KUKA KRL program: MyProgram_253().src

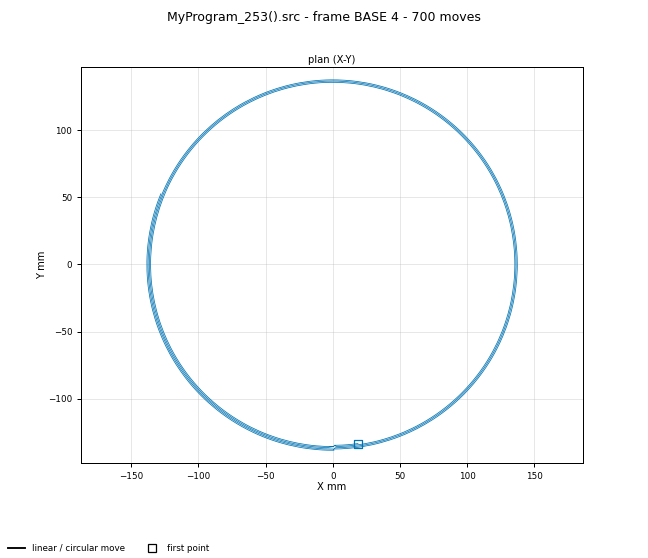
[picture p0: tool path of MyProgram_253().src in frame BASE 4, 700 of 700 moves have a stored position in this frame; points joined in program order, loops and branches not executed]
&ACCESS RVP
&REL 1
&PARAM TEMPLATE = C:\KRC\Roboter\Template\vorgabe
&PARAM EDITMASK = *
DEF MyProgram_253()
; ---- Setting reference (Base) ----
$BASE = BASE_DATA[4]

; --------------------------
; ---- Setting tool (TCP) ----
$TOOL = TOOL_DATA[3]
; --------------------------

$VEL.CP = VEL_APROX_PRINT
Startdeposition()
$VEL.CP = VEL_PRINT
LIN {X 18.8097,Y -133.4108,Z 165,A -80.9868,B 11.6438,C 0.2776,E1 11.6692,E2 531.5749} C_DIS
LIN {X 14.6629,Y -133.9301,Z 165,A -82.8153,B 11.6437,C 0.2797,E1 11.6641,E2 533.4109} C_DIS
LIN {X 11.2061,Y -134.2633,Z 165,A -84.2006,B 11.6437,C 0.278,E1 11.6603,E2 534.7857} C_DIS
LIN {X 7.424,Y -134.5271,Z 165,A -85.9426,B 11.6437,C 0.2818,E1 11.6554,E2 536.5447} C_DIS
LIN {X 3.6896,Y -134.6797,Z 165,A -87.3882,B 11.6437,C 0.2785,E1 11.6514,E2 537.9732} C_DIS
LIN {X 0.9754,Y -134.7225,Z 165,A -88.2258,B 11.6439,C 0.2708,E1 11.6492,E2 538.7721} C_DIS
Enddeposition()
LIN {X 0.9754,Y -134.7225,Z 165,A -88.2258,B 11.6439,C 0.2708,E1 11.6492,E2 538.7721} C_DIS
Startdeposition()
$VEL.CP = VEL_PRINT
LIN {X 3.0109,Y -135.617,Z 165,A -86.906,B 11.5615,C 0.2702,E1 11.5704,E2 537.4539} C_DIS
LIN {X 6.5276,Y -135.4914,Z 165,A -85.4969,B 11.5615,C 0.2718,E1 11.5743,E2 536.0536} C_DIS
LIN {X 10.0387,Y -135.2764,Z 165,A -84.0037,B 11.5615,C 0.2711,E1 11.5785,E2 534.5587} C_DIS
LIN {X 14.2252,Y -134.9006,Z 165,A -82.4774,B 11.5613,C 0.2767,E1 11.5827,E2 533.0628} C_DIS
LIN {X 17.3372,Y -134.536,Z 165,A -80.9699,B 11.5615,C 0.2714,E1 11.5869,E2 531.5314} C_DIS
LIN {X 20.6164,Y -134.0724,Z 165,A -79.5566,B 11.5615,C 0.2702,E1 11.5908,E2 530.1154} C_DIS
LIN {X 24.6834,Y -133.3858,Z 165,A -77.688,B 11.5615,C 0.2658,E1 11.596,E2 528.2297} C_DIS
LIN {X 27.8368,Y -132.7635,Z 165,A -76.3315,B 11.5616,C 0.2649,E1 11.5997,E2 526.8724} C_DIS
LIN {X 30.9968,Y -132.0615,Z 165,A -74.966,B 11.5616,C 0.2638,E1 11.6034,E2 525.5062} C_DIS
LIN {X 34.1606,Y -131.2787,Z 165,A -73.7387,B 11.5616,C 0.2666,E1 11.6067,E2 524.2967} C_DIS
LIN {X 37.6859,Y -130.3086,Z 165,A -72.3391,B 11.5616,C 0.2689,E1 11.6104,E2 522.9142} C_DIS
LIN {X 40.9847,Y -129.3086,Z 165,A -70.9423,B 11.5616,C 0.269,E1 11.6141,E2 521.5237} C_DIS
LIN {X 43.6454,Y -128.4373,Z 165,A -69.4187,B 11.5617,C 0.2588,E1 11.6183,E2 519.9563} C_DIS
LIN {X 47.2884,Y -127.1387,Z 165,A -67.9407,B 11.5617,C 0.261,E1 11.6221,E2 518.4965} C_DIS
LIN {X 49.9322,Y -126.1262,Z 165,A -66.7499,B 11.5617,C 0.2598,E1 11.6252,E2 517.3055} C_DIS
LIN {X 53.0552,Y -124.8446,Z 165,A -65.3304,B 11.5617,C 0.2581,E1 11.6289,E2 515.8856} C_DIS
LIN {X 56.4766,Y -123.3327,Z 165,A -63.8884,B 11.5617,C 0.2597,E1 11.6325,E2 514.4594} C_DIS
LIN {X 59.2442,Y -122.0294,Z 165,A -62.4727,B 11.5618,C 0.2546,E1 11.6361,E2 513.0272} C_DIS
LIN {X 62.3035,Y -120.4961,Z 165,A -60.97,B 11.5619,C 0.251,E1 11.6399,E2 511.5159} C_DIS
LIN {X 66.0881,Y -118.4627,Z 165,A -59.1023,B 11.562,C 0.2468,E1 11.6445,E2 509.6398} C_DIS
LIN {X 69.8227,Y -116.3006,Z 165,A -57.2966,B 11.562,C 0.2443,E1 11.6488,E2 507.8345} C_DIS
LIN {X 73.5009,Y -114.0116,Z 165,A -55.5367,B 11.562,C 0.2431,E1 11.6529,E2 506.0816} C_DIS
LIN {X 77.1164,Y -111.598,Z 165,A -53.6553,B 11.5622,C 0.2386,E1 11.6573,E2 504.1927} C_DIS
LIN {X 80.6628,Y -109.0622,Z 165,A -51.8858,B 11.5622,C 0.2372,E1 11.6613,E2 502.4305} C_DIS
LIN {X 84.1341,Y -106.4072,Z 165,A -50.0545,B 11.5622,C 0.2341,E1 11.6653,E2 500.5991} C_DIS
LIN {X 87.5243,Y -103.6366,Z 165,A -48.1855,B 11.5624,C 0.2299,E1 11.6693,E2 498.7257} C_DIS
LIN {X 90.8278,Y -100.7539,Z 165,A -46.385,B 11.5624,C 0.2275,E1 11.6731,E2 496.9297} C_DIS
LIN {X 93.8395,Y -97.9542,Z 165,A -44.6945,B 11.5624,C 0.2251,E1 11.6765,E2 495.2431} C_DIS
LIN {X 96.5381,Y -95.2966,Z 165,A -43.0391,B 11.5625,C 0.2201,E1 11.6798,E2 493.579} C_DIS
LIN {X 99.5704,Y -92.1237,Z 165,A -41.3104,B 11.5625,C 0.2194,E1 11.6831,E2 491.8641} C_DIS
LIN {X 101.9202,Y -89.5172,Z 165,A -39.7769,B 11.5626,C 0.2146,E1 11.6859,E2 490.3225} C_DIS
LIN {X 104.7585,Y -86.1783,Z 165,A -37.8873,B 11.5627,C 0.2092,E1 11.6893,E2 488.4259} C_DIS
LIN {X 107.563,Y -82.6508,Z 165,A -36.0363,B 11.5627,C 0.206,E1 11.6925,E2 486.5794} C_DIS
LIN {X 110.091,Y -79.2529,Z 165,A -34.2361,B 11.5629,C 0.2013,E1 11.6955,E2 484.7757} C_DIS
LIN {X 112.5783,Y -75.6781,Z 165,A -32.4181,B 11.5629,C 0.1973,E1 11.6983,E2 482.9583} C_DIS
LIN {X 115.0446,Y -71.8725,Z 165,A -30.6305,B 11.5629,C 0.196,E1 11.701,E2 481.1846} C_DIS
LIN {X 117.1808,Y -68.3353,Z 165,A -28.8018,B 11.5631,C 0.1892,E1 11.7036,E2 479.3433} C_DIS
LIN {X 119.3066,Y -64.552,Z 165,A -27.0042,B 11.5631,C 0.1853,E1 11.706,E2 477.5481} C_DIS
LIN {X 120.7405,Y -61.8235,Z 165,A -25.8285,B 11.5631,C 0.1853,E1 11.7075,E2 476.3866} C_DIS
LIN {X 122.2606,Y -58.7602,Z 165,A -24.4024,B 11.5631,C 0.182,E1 11.7093,E2 474.9612} C_DIS
LIN {X 123.609,Y -55.8697,Z 165,A -23.1901,B 11.5631,C 0.182,E1 11.7107,E2 473.7643} C_DIS
LIN {X 125.0285,Y -52.615,Z 165,A -21.5784,B 11.5633,C 0.1748,E1 11.7125,E2 472.1368} C_DIS
LIN {X 126.1262,Y -49.9322,Z 165,A -20.3839,B 11.5633,C 0.1722,E1 11.7137,E2 470.9447} C_DIS
LIN {X 127.3237,Y -46.7945,Z 165,A -18.8366,B 11.5634,C 0.1646,E1 11.7152,E2 469.3796} C_DIS
LIN {X 128.6025,Y -43.1491,Z 165,A -17.5683,B 11.5634,C 0.1702,E1 11.7163,E2 468.1549} C_DIS
LIN {X 129.6194,Y -39.9908,Z 165,A -15.9931,B 11.5634,C 0.1614,E1 11.7177,E2 466.5564} C_DIS
LIN {X 130.5534,Y -36.8277,Z 165,A -14.6194,B 11.5635,C 0.1579,E1 11.7187,E2 465.1834} C_DIS
LIN {X 131.2787,Y -34.1606,Z 165,A -13.3235,B 11.5636,C 0.151,E1 11.7197,E2 463.8702} C_DIS
LIN {X 132.0615,Y -30.9968,Z 165,A -11.9672,B 11.5636,C 0.1476,E1 11.7206,E2 462.515} C_DIS
LIN {X 132.8446,Y -27.4386,Z 165,A -10.5679,B 11.5636,C 0.147,E1 11.7214,E2 461.1313} C_DIS
LIN {X 133.4744,Y -24.1886,Z 165,A -9.216,B 11.5637,C 0.1442,E1 11.722,E2 459.7837} C_DIS
LIN {X 133.9295,Y -21.5393,Z 165,A -8.0963,B 11.5637,C 0.1414,E1 11.7226,E2 458.6648} C_DIS
LIN {X 134.4521,Y -17.9776,Z 165,A -6.5824,B 11.5638,C 0.1371,E1 11.7231,E2 457.1498} C_DIS
LIN {X 134.8403,Y -14.7856,Z 165,A -5.2517,B 11.5638,C 0.1338,E1 11.7236,E2 455.8211} C_DIS
LIN {X 135.2321,Y -10.6455,Z 165,A -3.393,B 11.5639,C 0.1258,E1 11.724,E2 453.9477} C_DIS
LIN {X 135.4388,Y -7.5745,Z 165,A -2.248,B 11.5639,C 0.1263,E1 11.7242,E2 452.8208} C_DIS
LIN {X 135.5882,Y -4.0496,Z 165,A -0.7384,B 11.5639,C 0.1214,E1 11.7244,E2 451.307} C_DIS
LIN {X 135.6518,Y -0.0881,Z 165,A 0.931,B 11.564,C 0.1166,E1 11.7244,E2 449.6365} C_DIS
LIN {X 135.617,Y 3.0109,Z 165,A 2.3297,B 11.564,C 0.1102,E1 11.7244,E2 448.2252} C_DIS
LIN {X 135.4388,Y 7.5745,Z 165,A 4.2095,B 11.5641,C 0.1059,E1 11.7241,E2 446.3495} C_DIS
LIN {X 135.1735,Y 11.3391,Z 165,A 5.6788,B 11.5641,C 0.1047,E1 11.7238,E2 444.8941} C_DIS
LIN {X 134.786,Y 15.2895,Z 165,A 7.4472,B 11.5642,C 0.0972,E1 11.7232,E2 443.1126} C_DIS
LIN {X 134.3255,Y 18.8991,Z 165,A 8.828,B 11.5642,C 0.0972,E1 11.7227,E2 441.7497} C_DIS
LIN {X 133.9295,Y 21.5393,Z 165,A 10.076,B 11.5642,C 0.0905,E1 11.7222,E2 440.4858} C_DIS
LIN {X 133.3259,Y 24.9967,Z 165,A 11.4669,B 11.5642,C 0.0888,E1 11.7215,E2 439.1048} C_DIS
LIN {X 132.7036,Y 28.1146,Z 165,A 12.7978,B 11.5642,C 0.0853,E1 11.7207,E2 437.7741} C_DIS
LIN {X 131.9194,Y 31.5863,Z 165,A 14.2211,B 11.5643,C 0.0832,E1 11.7198,E2 436.3594} C_DIS
LIN {X 130.8567,Y 35.7431,Z 165,A 16.0164,B 11.5643,C 0.0786,E1 11.7186,E2 434.5646} C_DIS
LIN {X 129.9511,Y 38.9071,Z 165,A 17.5386,B 11.5643,C 0.071,E1 11.7173,E2 433.0247} C_DIS
LIN {X 128.9627,Y 42.0675,Z 165,A 18.8807,B 11.5644,C 0.0687,E1 11.7162,E2 431.6885} C_DIS
LIN {X 127.7125,Y 45.716,Z 165,A 20.3863,B 11.5644,C 0.0676,E1 11.7148,E2 430.1967} C_DIS
LIN {X 126.5438,Y 48.8579,Z 165,A 21.5904,B 11.5644,C 0.0696,E1 11.7137,E2 429.0177} C_DIS
LIN {X 125.4959,Y 51.4958,Z 165,A 22.9728,B 11.5644,C 0.0613,E1 11.7122,E2 427.6118} C_DIS
LIN {X 124.009,Y 54.9753,Z 165,A 24.592,B 11.5644,C 0.0564,E1 11.7104,E2 425.9886} C_DIS
LIN {X 122.7647,Y 57.7051,Z 165,A 25.8078,B 11.5644,C 0.0545,E1 11.709,E2 424.7782} C_DIS
LIN {X 121.1879,Y 60.9446,Z 165,A 27.3539,B 11.5644,C 0.0499,E1 11.707,E2 423.228} C_DIS
LIN {X 119.4381,Y 64.3071,Z 165,A 28.94,B 11.5645,C 0.0462,E1 11.705,E2 421.6426} C_DIS
LIN {X 117.3168,Y 68.1004,Z 165,A 30.7505,B 11.5645,C 0.0422,E1 11.7025,E2 419.834} C_DIS
LIN {X 115.0863,Y 71.8055,Z 165,A 32.5825,B 11.5645,C 0.0376,E1 11.6998,E2 418.0002} C_DIS
LIN {X 112.9044,Y 75.1896,Z 165,A 34.3027,B 11.5645,C 0.0329,E1 11.6971,E2 416.2765} C_DIS
LIN {X 110.2505,Y 79.0298,Z 165,A 36.1948,B 11.5645,C 0.0304,E1 11.6941,E2 414.393} C_DIS
LIN {X 107.8473,Y 82.279,Z 165,A 37.9476,B 11.5645,C 0.0252,E1 11.6912,E2 412.6336} C_DIS
LIN {X 105.1384,Y 85.7135,Z 165,A 39.7777,B 11.5645,C 0.0215,E1 11.688,E2 410.8047} C_DIS
LIN {X 102.11,Y 89.2997,Z 165,A 41.6814,B 11.5645,C 0.0193,E1 11.6845,E2 408.9098} C_DIS
LIN {X 99.3823,Y 92.3257,Z 165,A 43.4086,B 11.5645,C 0.0155,E1 11.6813,E2 407.181} C_DIS
LIN {X 96.4447,Y 95.3906,Z 165,A 45.241,B 11.5645,C 0.0107,E1 11.6777,E2 405.343} C_DIS
LIN {X 93.2037,Y 98.5594,Z 165,A 47.0833,B 11.5646,C 0.0088,E1 11.674,E2 403.5088} C_DIS
LIN {X 90.0627,Y 101.4379,Z 165,A 48.9007,B 11.5646,C 0.0049,E1 11.6702,E2 401.6886} C_DIS
LIN {X 86.853,Y 104.1998,Z 165,A 50.7053,B 11.5646,C 0.0011,E1 11.6664,E2 399.8814} C_DIS
LIN {X 83.4461,Y 106.9476,Z 165,A 52.5387,B 11.5646,C -0.0017,E1 11.6623,E2 398.0494} C_DIS
LIN {X 79.9593,Y 109.579,Z 165,A 54.3106,B 11.5646,C -0.0029,E1 11.6584,E2 396.286} C_DIS
LIN {X 76.3986,Y 112.0906,Z 165,A 56.195,B 11.5646,C -0.0071,E1 11.654,E2 394.3958} C_DIS
LIN {X 72.7701,Y 114.4795,Z 165,A 57.9895,B 11.5646,C -0.0089,E1 11.6498,E2 392.6059} C_DIS
LIN {X 69.0801,Y 116.7432,Z 165,A 59.7732,B 11.5646,C -0.0104,E1 11.6456,E2 390.8275} C_DIS
LIN {X 65.335,Y 118.8797,Z 165,A 61.6147,B 11.5646,C -0.0134,E1 11.6411,E2 388.9832} C_DIS
LIN {X 61.8235,Y 120.7405,Z 165,A 63.1832,B 11.5646,C -0.0128,E1 11.6372,E2 387.428} C_DIS
LIN {X 58.7602,Y 122.2606,Z 165,A 64.6185,B 11.5646,C -0.0143,E1 11.6336,E2 385.9938} C_DIS
LIN {X 55.7713,Y 123.653,Z 165,A 65.996,B 11.5646,C -0.0156,E1 11.6302,E2 384.6182} C_DIS
LIN {X 53.0552,Y 124.8446,Z 165,A 67.2485,B 11.5646,C -0.0169,E1 11.6269,E2 383.3658} C_DIS
LIN {X 49.9322,Y 126.1262,Z 165,A 68.666,B 11.5646,C -0.0182,E1 11.6233,E2 381.9494} C_DIS
LIN {X 46.2991,Y 127.5023,Z 165,A 70.2974,B 11.5646,C -0.0196,E1 11.619,E2 380.3191} C_DIS
LIN {X 43.1491,Y 128.6025,Z 165,A 71.5042,B 11.5646,C -0.0157,E1 11.6159,E2 379.1371} C_DIS
LIN {X 39.9908,Y 129.6194,Z 165,A 73.0939,B 11.5646,C -0.0217,E1 11.6116,E2 377.5247} C_DIS
LIN {X 36.8277,Y 130.5534,Z 165,A 74.4804,B 11.5646,C -0.0225,E1 11.6079,E2 376.1392} C_DIS
LIN {X 33.5566,Y 131.432,Z 165,A 75.8775,B 11.5646,C -0.0227,E1 11.6041,E2 374.7464} C_DIS
LIN {X 30.9968,Y 132.0615,Z 165,A 77.159,B 11.5646,C -0.0276,E1 11.6006,E2 373.4448} C_DIS
LIN {X 27.2576,Y 132.8814,Z 165,A 78.6291,B 11.5646,C -0.0248,E1 11.5966,E2 371.9929} C_DIS
LIN {X 24.0786,Y 133.494,Z 165,A 79.9581,B 11.5646,C -0.0245,E1 11.593,E2 370.669} C_DIS
LIN {X 19.9716,Y 134.1722,Z 165,A 81.7388,B 11.5646,C -0.0258,E1 11.5881,E2 368.8862} C_DIS
LIN {X 16.3568,Y 134.6587,Z 165,A 83.3166,B 11.5646,C -0.0272,E1 11.5837,E2 367.3043} C_DIS
LIN {X 12.9514,Y 135.0285,Z 165,A 84.5827,B 11.5646,C -0.0231,E1 11.5802,E2 366.0606} C_DIS
LIN {X 8.6253,Y 135.3741,Z 165,A 86.3643,B 11.5646,C -0.0222,E1 11.5753,E2 364.2859} C_DIS
LIN {X 6.0473,Y 135.5156,Z 165,A 87.7701,B 11.5646,C -0.03,E1 11.5712,E2 362.8424} C_DIS
LIN {X 2.2479,Y 135.6297,Z 165,A 89.2777,B 11.5646,C -0.0276,E1 11.5671,E2 361.3474} C_DIS
LIN {X -1.5021,Y 135.6421,Z 165,A 90.821,B 11.5646,C -0.0265,E1 11.5628,E2 359.8098} C_DIS
LIN {X -5.0045,Y 135.5563,Z 165,A 92.3049,B 11.5646,C -0.0265,E1 11.5586,E2 358.3261} C_DIS
LIN {X -9.5911,Y 135.3091,Z 165,A 94.2998,B 11.5646,C -0.0273,E1 11.5531,E2 356.3256} C_DIS
LIN {X -13.0285,Y 135.0211,Z 165,A 95.7196,B 11.5646,C -0.0259,E1 11.5491,E2 354.9111} C_DIS
LIN {X -16.3568,Y 134.6587,Z 165,A 97.1764,B 11.5646,C -0.0264,E1 11.5451,E2 353.4499} C_DIS
LIN {X -20.4646,Y 134.0959,Z 165,A 98.701,B 11.5646,C -0.0201,E1 11.5409,E2 351.9539} C_DIS
LIN {X -23.5279,Y 133.5926,Z 165,A 100.0547,B 11.5646,C -0.0204,E1 11.5372,E2 350.5958} C_DIS
LIN {X -26.7552,Y 132.9836,Z 165,A 101.4078,B 11.5646,C -0.0188,E1 11.5335,E2 349.2478} C_DIS
LIN {X -29.9133,Y 132.309,Z 165,A 102.9616,B 11.5646,C -0.0223,E1 11.5292,E2 347.672} C_DIS
LIN {X -33.154,Y 131.5342,Z 165,A 104.3866,B 11.5646,C -0.0217,E1 11.5253,E2 346.2458} C_DIS
LIN {X -37.3253,Y 130.4142,Z 165,A 106.2181,B 11.5646,C -0.0203,E1 11.5204,E2 344.4148} C_DIS
LIN {X -40.9847,Y 129.3086,Z 165,A 107.6438,B 11.5646,C -0.0144,E1 11.5167,E2 343.0131} C_DIS
LIN {X -43.6454,Y 128.4373,Z 165,A 109.1827,B 11.5646,C -0.0216,E1 11.5125,E2 341.4321} C_DIS
LIN {X -47.2884,Y 127.1387,Z 165,A 110.694,B 11.5646,C -0.017,E1 11.5086,E2 339.9369} C_DIS
LIN {X -50.0761,Y 126.0682,Z 165,A 112.0495,B 11.5646,C -0.0177,E1 11.505,E2 338.571} C_DIS
LIN {X -53.5443,Y 124.6332,Z 165,A 113.5395,B 11.5646,C -0.0136,E1 11.5012,E2 337.0939} C_DIS
LIN {X -56.1603,Y 123.479,Z 165,A 114.8903,B 11.5646,C -0.0154,E1 11.4977,E2 335.7268} C_DIS
LIN {X -59.6227,Y 121.8427,Z 165,A 116.2236,B 11.5646,C -0.0067,E1 11.4945,E2 334.4294} C_DIS
LIN {X -62.3035,Y 120.4961,Z 165,A 117.7264,B 11.5646,C -0.0103,E1 11.4906,E2 332.8992} C_DIS
LIN {X -66.0881,Y 118.4627,Z 165,A 119.6134,B 11.5646,C -0.0093,E1 11.486,E2 331.005} C_DIS
LIN {X -69.8227,Y 116.3006,Z 165,A 121.4506,B 11.5646,C -0.0068,E1 11.4816,E2 329.1679} C_DIS
LIN {X -73.5009,Y 114.0116,Z 165,A 123.2364,B 11.5646,C -0.0029,E1 11.4774,E2 327.3892} C_DIS
LIN {X -77.1164,Y 111.598,Z 165,A 125.1472,B 11.5646,C -0.0014,E1 11.473,E2 325.471} C_DIS
LIN {X -80.782,Y 108.9734,Z 165,A 126.9705,B 11.5646,C 0.0038,E1 11.4689,E2 323.6595} C_DIS
LIN {X -84.1341,Y 106.4072,Z 165,A 128.8073,B 11.5646,C 0.0059,E1 11.4648,E2 321.818} C_DIS
LIN {X -87.5243,Y 103.6366,Z 165,A 130.7206,B 11.5646,C 0.008,E1 11.4607,E2 319.8989} C_DIS
LIN {X -90.9093,Y 100.6799,Z 165,A 132.5608,B 11.5646,C 0.0131,E1 11.4569,E2 318.0676} C_DIS
LIN {X -93.8395,Y 97.9542,Z 165,A 134.2643,B 11.5646,C 0.0163,E1 11.4534,E2 316.3643} C_DIS
LIN {X -96.5381,Y 95.2966,Z 165,A 135.9106,B 11.5646,C 0.0187,E1 11.4502,E2 314.7141} C_DIS
LIN {X -99.5589,Y 92.136,Z 165,A 137.8243,B 11.5646,C 0.0213,E1 11.4465,E2 312.7943} C_DIS
LIN {X -102.4967,Y 88.8564,Z 165,A 139.7132,B 11.5646,C 0.0248,E1 11.443,E2 310.9038} C_DIS
LIN {X -105.3127,Y 85.5002,Z 165,A 141.5823,B 11.5646,C 0.0287,E1 11.4397,E2 309.0346} C_DIS
LIN {X -108.0143,Y 82.0606,Z 165,A 143.4486,B 11.5646,C 0.0327,E1 11.4365,E2 307.1681} C_DIS
LIN {X -110.5982,Y 78.5436,Z 165,A 145.2536,B 11.5646,C 0.038,E1 11.4336,E2 305.3698} C_DIS
LIN {X -113.061,Y 74.955,Z 165,A 147.1093,B 11.5646,C 0.0422,E1 11.4307,E2 303.514} C_DIS
LIN {X -115.4001,Y 71.3011,Z 165,A 148.9614,B 11.5646,C 0.0464,E1 11.4279,E2 301.6617} C_DIS
LIN {X -117.6132,Y 67.5883,Z 165,A 150.8065,B 11.5645,C 0.0507,E1 11.4253,E2 299.8163} C_DIS
LIN {X -119.7002,Y 63.8193,Z 165,A 152.5779,B 11.5645,C 0.0565,E1 11.423,E2 298.0529} C_DIS
LIN {X -121.2732,Y 60.7771,Z 165,A 154.0421,B 11.5645,C 0.06,E1 11.4211,E2 296.5882} C_DIS
LIN {X -122.7647,Y 57.7051,Z 165,A 155.5007,B 11.5645,C 0.0635,E1 11.4194,E2 295.1294} C_DIS
LIN {X -124.1723,Y 54.6102,Z 165,A 156.9527,B 11.5645,C 0.0671,E1 11.4177,E2 293.677} C_DIS
LIN {X -125.6284,Y 51.1672,Z 165,A 158.4145,B 11.5644,C 0.0739,E1 11.4161,E2 292.2312} C_DIS
LIN {X -126.7354,Y 48.365,Z 165,A 159.8366,B 11.5644,C 0.0743,E1 11.4147,E2 290.7925} C_DIS
LIN {X -128.0627,Y 44.7256,Z 165,A 161.4909,B 11.5644,C 0.0784,E1 11.4131,E2 289.1378} C_DIS
LIN {X -128.9627,Y 42.0675,Z 165,A 162.8416,B 11.5644,C 0.0782,E1 11.4119,E2 287.7683} C_DIS
LIN {X -130.1232,Y 38.3193,Z 165,A 164.3422,B 11.5643,C 0.0863,E1 11.4107,E2 286.2887} C_DIS
LIN {X -130.9894,Y 35.2454,Z 165,A 165.5349,B 11.5643,C 0.0935,E1 11.4099,E2 285.1166} C_DIS
LIN {X -131.8001,Y 32.0811,Z 165,A 166.9315,B 11.5643,C 0.0971,E1 11.4089,E2 283.7195} C_DIS
LIN {X -132.5298,Y 28.9195,Z 165,A 168.5512,B 11.5643,C 0.0957,E1 11.4079,E2 282.071} C_DIS
LIN {X -133.1793,Y 25.7636,Z 165,A 169.889,B 11.5642,C 0.1002,E1 11.4072,E2 280.7375} C_DIS
LIN {X -133.7541,Y 22.5907,Z 165,A 171.0669,B 11.5642,C 0.1081,E1 11.4066,E2 279.5837} C_DIS
LIN {X -134.1722,Y 19.9716,Z 165,A 172.4004,B 11.5642,C 0.1068,E1 11.406,E2 278.2255} C_DIS
LIN {X -134.6587,Y 16.3568,Z 165,A 173.9948,B 11.5641,C 0.1102,E1 11.4055,E2 276.6261} C_DIS
LIN {X -135.1017,Y 12.1888,Z 165,A 175.7494,B 11.5641,C 0.1157,E1 11.405,E2 274.8755} C_DIS
LIN {X -135.3741,Y 8.6253,Z 165,A 177.3068,B 11.564,C 0.1191,E1 11.4047,E2 273.3138} C_DIS
LIN {X -135.5381,Y 5.4688,Z 165,A 178.6286,B 11.564,C 0.1234,E1 11.4045,E2 271.995} C_DIS
LIN {X -135.6273,Y 2.3909,Z 165,A 179.9187,B 11.564,C 0.1274,E1 11.4045,E2 270.7077} C_DIS
LIN {X -135.6421,Y -1.5021,Z 165,A -178.3918,B 11.5639,C 0.1313,E1 11.4045,E2 269.0145} C_DIS
LIN {X -135.5563,Y -5.0045,Z 165,A -176.8629,B 11.5639,C 0.1346,E1 11.4045,E2 267.481} C_DIS
LIN {X -135.397,Y -8.2536,Z 165,A -175.4646,B 11.5638,C 0.1381,E1 11.4048,E2 266.0811} C_DIS
LIN {X -135.1501,Y -11.6162,Z 165,A -173.9891,B 11.5638,C 0.1412,E1 11.4051,E2 264.6008} C_DIS
LIN {X -134.7755,Y -15.3779,Z 165,A -172.3118,B 11.5638,C 0.1441,E1 11.4056,E2 262.9152} C_DIS
LIN {X -134.3255,Y -18.8991,Z 165,A -170.9059,B 11.5636,C 0.1505,E1 11.4061,E2 261.5223} C_DIS
LIN {X -133.9295,Y -21.5393,Z 165,A -169.7004,B 11.5636,C 0.1521,E1 11.4067,E2 260.3083} C_DIS
LIN {X -133.3858,Y -24.6834,Z 165,A -168.2475,B 11.5636,C 0.1537,E1 11.4074,E2 258.8439} C_DIS
LIN {X -132.7635,Y -27.8368,Z 165,A -166.8584,B 11.5636,C 0.1569,E1 11.4082,E2 257.4521} C_DIS
LIN {X -131.9958,Y -31.2695,Z 165,A -165.4457,B 11.5635,C 0.1627,E1 11.4091,E2 256.0498} C_DIS
LIN {X -131.2787,Y -34.1606,Z 165,A -164.234,B 11.5635,C 0.1673,E1 11.4099,E2 254.845} C_DIS
LIN {X -130.4142,Y -37.3253,Z 165,A -162.8288,B 11.5634,C 0.1707,E1 11.411,E2 253.4386} C_DIS
LIN {X -129.3086,Y -40.9847,Z 165,A -161.22,B 11.5633,C 0.1753,E1 11.4123,E2 251.8319} C_DIS
LIN {X -128.2806,Y -44.0971,Z 165,A -159.7755,B 11.5633,C 0.1779,E1 11.4136,E2 250.3811} C_DIS
LIN {X -127.1387,Y -47.2884,Z 165,A -158.3369,B 11.5632,C 0.1816,E1 11.4149,E2 248.9429} C_DIS
LIN {X -126.1262,Y -49.9322,Z 165,A -156.9762,B 11.5632,C 0.1812,E1 11.4164,E2 247.5628} C_DIS
LIN {X -124.6332,Y -53.5443,Z 165,A -155.4525,B 11.5631,C 0.1884,E1 11.418,E2 246.0561} C_DIS
LIN {X -123.479,Y -56.1603,Z 165,A -154.2295,B 11.5631,C 0.1913,E1 11.4194,E2 244.8323} C_DIS
LIN {X -121.8678,Y -59.5718,Z 165,A -152.7548,B 11.5629,C 0.1981,E1 11.4212,E2 243.3734} C_DIS
LIN {X -120.4961,Y -62.3035,Z 165,A -151.2417,B 11.5629,C 0.1965,E1 11.4231,E2 241.8339} C_DIS
LIN {X -118.4627,Y -66.0881,Z 165,A -149.3458,B 11.5629,C 0.1993,E1 11.4257,E2 239.9291} C_DIS
LIN {X -116.3006,Y -69.8227,Z 165,A -147.501,B 11.5629,C 0.2033,E1 11.4283,E2 238.0829} C_DIS
LIN {X -113.9537,Y -73.5901,Z 165,A -145.6908,B 11.5627,C 0.2093,E1 11.431,E2 236.2818} C_DIS
LIN {X -111.598,Y -77.1164,Z 165,A -143.7923,B 11.5627,C 0.2112,E1 11.434,E2 234.3712} C_DIS
LIN {X -109.0064,Y -80.7377,Z 165,A -141.9744,B 11.5626,C 0.2169,E1 11.437,E2 232.5621} C_DIS
LIN {X -106.4072,Y -84.1341,Z 165,A -140.1246,B 11.5626,C 0.22,E1 11.4401,E2 230.708} C_DIS
LIN {X -103.6366,Y -87.5243,Z 165,A -138.2565,B 11.5625,C 0.2237,E1 11.4435,E2 228.8385} C_DIS
LIN {X -100.7998,Y -90.7766,Z 165,A -136.4082,B 11.5625,C 0.227,E1 11.4469,E2 226.9879} C_DIS
LIN {X -97.9542,Y -93.8395,Z 165,A -134.6601,B 11.5623,C 0.231,E1 11.4502,E2 225.2428} C_DIS
LIN {X -94.8669,Y -96.9595,Z 165,A -132.7938,B 11.5623,C 0.2344,E1 11.4539,E2 223.3758} C_DIS
LIN {X -91.6889,Y -99.9701,Z 165,A -130.9272,B 11.5622,C 0.2376,E1 11.4578,E2 221.5076} C_DIS
LIN {X -88.6475,Y -102.6766,Z 165,A -129.1318,B 11.5622,C 0.239,E1 11.4615,E2 219.7033} C_DIS
LIN {X -85.0331,Y -105.6894,Z 165,A -127.1509,B 11.5621,C 0.2427,E1 11.4658,E2 217.7239} C_DIS
LIN {X -81.5826,Y -108.3751,Z 165,A -125.3326,B 11.5621,C 0.2464,E1 11.4698,E2 215.9096} C_DIS
LIN {X -78.0814,Y -110.9242,Z 165,A -123.4857,B 11.562,C 0.249,E1 11.474,E2 214.061} C_DIS
LIN {X -74.4575,Y -113.3886,Z 165,A -121.6284,B 11.562,C 0.2517,E1 11.4784,E2 212.2033} C_DIS
LIN {X -71.069,Y -115.5425,Z 165,A -119.8599,B 11.5619,C 0.2524,E1 11.4826,E2 210.426} C_DIS
LIN {X -67.0385,Y -117.9268,Z 165,A -117.9408,B 11.5618,C 0.2565,E1 11.4872,E2 208.5145} C_DIS
LIN {X -63.8229,Y -119.6983,Z 165,A -116.4117,B 11.5618,C 0.2591,E1 11.4909,E2 206.9882} C_DIS
LIN {X -60.7771,Y -121.2732,Z 165,A -114.9567,B 11.5618,C 0.2607,E1 11.4946,E2 205.5325} C_DIS
LIN {X -57.4109,Y -122.9007,Z 165,A -113.493,B 11.5616,C 0.2652,E1 11.4982,E2 204.0832} C_DIS
LIN {X -54.6102,Y -124.1723,Z 165,A -112.0668,B 11.5616,C 0.2636,E1 11.5019,E2 202.6412} C_DIS
LIN {X -51.4958,Y -125.4959,Z 165,A -110.4839,B 11.5616,C 0.2614,E1 11.506,E2 201.039} C_DIS
LIN {X -48.1022,Y -126.8339,Z 165,A -109.1927,B 11.5616,C 0.2688,E1 11.5093,E2 199.7789} C_DIS
LIN {X -44.7256,Y -128.0627,Z 165,A -107.5659,B 11.5616,C 0.2675,E1 11.5136,E2 198.1383} C_DIS
LIN {X -42.0675,Y -128.9627,Z 165,A -106.2281,B 11.5616,C 0.2648,E1 11.5172,E2 196.7813} C_DIS
LIN {X -38.4097,Y -130.0967,Z 165,A -104.7571,B 11.5616,C 0.2695,E1 11.5211,E2 195.3284} C_DIS
LIN {X -35.2454,Y -130.9894,Z 165,A -103.5594,B 11.5614,C 0.2751,E1 11.5243,E2 194.1544} C_DIS
LIN {X -32.0811,Y -131.8001,Z 165,A -101.9595,B 11.5614,C 0.2705,E1 11.5287,E2 192.5267} C_DIS
LIN {X -28.8513,Y -132.5445,Z 165,A -100.5992,B 11.5614,C 0.2722,E1 11.5324,E2 191.171} C_DIS
LIN {X -25.7636,Y -133.1793,Z 165,A -99.2518,B 11.5614,C 0.2724,E1 11.5361,E2 189.8213} C_DIS
LIN {X -22.616,Y -133.7498,Z 165,A -98.0879,B 11.5614,C 0.2775,E1 11.5392,E2 188.6805} C_DIS
LIN {X -19.4435,Y -134.2477,Z 165,A -96.5348,B 11.5614,C 0.2731,E1 11.5436,E2 187.1022} C_DIS
LIN {X -15.2758,Y -134.7875,Z 165,A -94.6349,B 11.5614,C 0.2704,E1 11.5489,E2 185.1862} C_DIS
LIN {X -12.1888,Y -135.1017,Z 165,A -93.461,B 11.5614,C 0.274,E1 11.5521,E2 184.029} C_DIS
LIN {X -8.6253,Y -135.3741,Z 165,A -92.1348,B 11.5613,C 0.2787,E1 11.5557,E2 182.7251} C_DIS
LIN {X -6.0473,Y -135.5156,Z 165,A -90.72,B 11.5615,C 0.2706,E1 11.5598,E2 181.2691} C_DIS
LIN {X -2.5364,Y -135.6249,Z 165,A -89.3856,B 11.5614,C 0.2742,E1 11.5634,E2 179.9528} C_DIS
LIN {X 0.9805,Y -135.645,Z 165,A -88.2691,B 11.5612,C 0.2833,E1 11.5664,E2 178.8818} C_DIS
Enddeposition()
LIN {X 0.9805,Y -135.645,Z 165,A -88.2691,B 11.5612,C 0.2833,E1 11.5664,E2 178.8818} C_DIS
Startdeposition()
$VEL.CP = VEL_PRINT
LIN {X -4.8472,Y -136.4812,Z 165,A -90.7493,B 11.4776,C 0.2955,E1 11.4761,E2 181.4277} C_DIS
LIN {X -12.6494,Y -135.9799,Z 165,A -94.4973,B 11.4773,C 0.3069,E1 11.4655,E2 185.2356} C_DIS
LIN {X -16.039,Y -135.6213,Z 165,A -95.3359,B 11.4777,C 0.292,E1 11.4633,E2 186.0006} C_DIS
LIN {X -18.8403,Y -135.2613,Z 165,A -96.9077,B 11.4774,C 0.3012,E1 11.4588,E2 187.6214} C_DIS
LIN {X -23.116,Y -134.5972,Z 165,A -98.9035,B 11.4774,C 0.305,E1 11.4533,E2 189.6404} C_DIS
LIN {X -26.3732,Y -133.9973,Z 165,A -99.9737,B 11.4775,C 0.2966,E1 11.4504,E2 190.6711} C_DIS
LIN {X -28.8971,Y -133.4739,Z 165,A -101.1058,B 11.4775,C 0.2973,E1 11.4473,E2 191.8097} C_DIS
LIN {X -32.0753,Y -132.746,Z 165,A -102.4528,B 11.4775,C 0.2961,E1 11.4437,E2 193.1543} C_DIS
LIN {X -35.8326,Y -131.7831,Z 165,A -104.0591,B 11.4775,C 0.2946,E1 11.4393,E2 194.7584} C_DIS
LIN {X -39.2032,Y -130.8206,Z 165,A -105.5408,B 11.4776,C 0.2938,E1 11.4354,E2 196.2417} C_DIS
LIN {X -41.863,Y -129.9918,Z 165,A -106.7854,B 11.4776,C 0.2947,E1 11.432,E2 197.496} C_DIS
LIN {X -45.23,Y -128.8596,Z 165,A -108.2308,B 11.4776,C 0.2924,E1 11.4282,E2 198.9359} C_DIS
LIN {X -48.9472,Y -127.4942,Z 165,A -109.7933,B 11.4777,C 0.2886,E1 11.4242,E2 200.4862} C_DIS
LIN {X -51.5608,Y -126.4596,Z 165,A -111.9329,B 11.4772,C 0.31,E1 11.4184,E2 202.7449} C_DIS
LIN {X -57.2369,Y -123.9927,Z 165,A -113.4053,B 11.4779,C 0.2808,E1 11.415,E2 204.0778} C_DIS
LIN {X -60.7798,Y -122.2956,Z 165,A -115.3661,B 11.4779,C 0.2862,E1 11.4099,E2 206.0778} C_DIS
LIN {X -64.2718,Y -120.4993,Z 165,A -117.0668,B 11.4779,C 0.2854,E1 11.4057,E2 207.785} C_DIS
LIN {X -68.0494,Y -118.4071,Z 165,A -118.9417,B 11.4779,C 0.2845,E1 11.4011,E2 209.6676} C_DIS
LIN {X -71.8922,Y -116.1137,Z 165,A -120.845,B 11.4779,C 0.2824,E1 11.3966,E2 211.5738} C_DIS
LIN {X -75.8191,Y -113.5881,Z 165,A -122.798,B 11.4779,C 0.2793,E1 11.392,E2 213.5257} C_DIS
LIN {X -79.5613,Y -110.9991,Z 165,A -124.6871,B 11.4781,C 0.2758,E1 11.3877,E2 215.4119} C_DIS
LIN {X -83.4797,Y -108.0832,Z 165,A -126.6501,B 11.4781,C 0.2704,E1 11.3833,E2 217.3637} C_DIS
LIN {X -86.5001,Y -105.6813,Z 165,A -129.106,B 11.4778,C 0.2865,E1 11.3778,E2 219.9224} C_DIS
LIN {X -91.0119,Y -101.8216,Z 165,A -130.7485,B 11.4784,C 0.2628,E1 11.3746,E2 221.4594} C_DIS
LIN {X -93.6995,Y -99.3538,Z 165,A -132.4653,B 11.4784,C 0.2641,E1 11.371,E2 223.1987} C_DIS
LIN {X -96.9974,Y -96.1369,Z 165,A -134.3985,B 11.4784,C 0.2602,E1 11.3672,E2 225.1312} C_DIS
LIN {X -100.0944,Y -92.9082,Z 165,A -136.2579,B 11.4785,C 0.256,E1 11.3636,E2 226.9876} C_DIS
LIN {X -102.8989,Y -89.7919,Z 165,A -138.1816,B 11.4785,C 0.256,E1 11.36,E2 228.9309} C_DIS
LIN {X -105.8587,Y -86.2829,Z 165,A -140.0123,B 11.4786,C 0.2496,E1 11.3568,E2 230.7488} C_DIS
LIN {X -108.6349,Y -82.7605,Z 165,A -141.9915,B 11.4786,C 0.2475,E1 11.3534,E2 232.739} C_DIS
LIN {X -111.0593,Y -79.4771,Z 165,A -143.6416,B 11.4788,C 0.2422,E1 11.3507,E2 234.3805} C_DIS
LIN {X -114.794,Y -73.9817,Z 165,A -146.4029,B 11.479,C 0.2349,E1 11.3464,E2 237.1368} C_DIS
LIN {X -117.0093,Y -70.4251,Z 165,A -148.2645,B 11.479,C 0.2329,E1 11.3437,E2 239.01} C_DIS
LIN {X -119.1931,Y -66.6625,Z 165,A -150.1036,B 11.479,C 0.2286,E1 11.3411,E2 240.8496} C_DIS
LIN {X -121.1489,Y -63.0352,Z 165,A -151.8182,B 11.4792,C 0.2239,E1 11.3389,E2 242.5612} C_DIS
LIN {X -123.2892,Y -58.7371,Z 165,A -153.7198,B 11.4793,C 0.2162,E1 11.3366,E2 244.4473} C_DIS
LIN {X -124.7479,Y -55.5719,Z 165,A -155.2796,B 11.4793,C 0.2145,E1 11.3348,E2 246.0181} C_DIS
LIN {X -126.1494,Y -52.3135,Z 165,A -156.7812,B 11.4794,C 0.2108,E1 11.3331,E2 247.5201} C_DIS
LIN {X -127.6329,Y -48.5864,Z 165,A -158.4899,B 11.4794,C 0.2068,E1 11.3314,E2 249.2307} C_DIS
LIN {X -129.3098,Y -43.9311,Z 165,A -160.5713,B 11.4796,C 0.2013,E1 11.3295,E2 251.3111} C_DIS
LIN {X -130.7476,Y -39.4418,Z 165,A -162.7082,B 11.4796,C 0.1992,E1 11.3277,E2 253.4657} C_DIS
LIN {X -132.5718,Y -32.7976,Z 165,A -165.4962,B 11.4798,C 0.1889,E1 11.3257,E2 256.2386} C_DIS
LIN {X -133.541,Y -28.5864,Z 165,A -167.3826,B 11.4798,C 0.1852,E1 11.3245,E2 258.1322} C_DIS
LIN {X -134.3577,Y -24.4647,Z 165,A -169.1685,B 11.4799,C 0.1807,E1 11.3236,E2 259.9194} C_DIS
LIN {X -134.9768,Y -20.7757,Z 165,A -170.7079,B 11.48,C 0.1755,E1 11.3229,E2 261.4535} C_DIS
LIN {X -135.4667,Y -17.3011,Z 165,A -172.3395,B 11.48,C 0.1746,E1 11.3223,E2 263.1032} C_DIS
LIN {X -135.943,Y -13.0334,Z 165,A -174.0606,B 11.4801,C 0.1676,E1 11.3218,E2 264.8126} C_DIS
LIN {X -136.2799,Y -8.8537,Z 165,A -175.8935,B 11.4801,C 0.1641,E1 11.3214,E2 266.6528} C_DIS
LIN {X -136.4695,Y -5.1481,Z 165,A -177.4143,B 11.4802,C 0.1587,E1 11.3212,E2 268.1676} C_DIS
LIN {X -136.5644,Y -0.8986,Z 165,A -179.1923,B 11.4803,C 0.1534,E1 11.3212,E2 269.9431} C_DIS
LIN {X -136.5493,Y 2.1701,Z 165,A 179.4903,B 11.4803,C 0.1502,E1 11.3212,E2 271.2628} C_DIS
LIN {X -136.4429,Y 5.8304,Z 165,A 177.7952,B 11.4803,C 0.149,E1 11.3213,E2 272.9756} C_DIS
LIN {X -136.1911,Y 10.1181,Z 165,A 176.0625,B 11.4805,C 0.1423,E1 11.3217,E2 274.6978} C_DIS
LIN {X -135.7777,Y 14.6558,Z 165,A 174.1672,B 11.4805,C 0.1363,E1 11.3222,E2 276.5891} C_DIS
LIN {X -135.3516,Y 18.1795,Z 165,A 172.7142,B 11.4805,C 0.1312,E1 11.3227,E2 278.0361} C_DIS
LIN {X -134.8482,Y 21.6062,Z 165,A 171.0511,B 11.4805,C 0.1314,E1 11.3234,E2 279.7232} C_DIS
LIN {X -134.1169,Y 25.7488,Z 165,A 169.3835,B 11.4807,C 0.1242,E1 11.3242,E2 281.3769} C_DIS
LIN {X -133.3971,Y 29.253,Z 165,A 167.7373,B 11.4807,C 0.1229,E1 11.3252,E2 283.0391} C_DIS
LIN {X -132.3955,Y 33.4926,Z 165,A 166.03,B 11.4807,C 0.1151,E1 11.3263,E2 284.7296} C_DIS
LIN {X -130.7572,Y 39.4104,Z 165,A 162.2663,B 11.4806,C 0.1327,E1 11.3294,E2 288.6332} C_DIS
LIN {X -128.3142,Y 46.7541,Z 165,A 160.0618,B 11.4809,C 0.1017,E1 11.3313,E2 290.709} C_DIS
LIN {X -126.4692,Y 51.5372,Z 165,A 157.9398,B 11.4809,C 0.0951,E1 11.3335,E2 292.825} C_DIS
LIN {X -125.2236,Y 54.4922,Z 165,A 156.5153,B 11.4809,C 0.0931,E1 11.3351,E2 294.2575} C_DIS
LIN {X -123.7181,Y 57.8307,Z 165,A 155.0476,B 11.4809,C 0.0875,E1 11.3368,E2 295.7151} C_DIS
LIN {X -122.379,Y 60.6108,Z 165,A 153.7048,B 11.481,C 0.0851,E1 11.3384,E2 297.0622} C_DIS
LIN {X -120.7512,Y 63.7927,Z 165,A 152.1885,B 11.481,C 0.0815,E1 11.3404,E2 298.5788} C_DIS
LIN {X -118.7375,Y 67.4704,Z 165,A 150.3071,B 11.481,C 0.0795,E1 11.3429,E2 300.4731} C_DIS
LIN {X -116.494,Y 71.2739,Z 165,A 148.447,B 11.481,C 0.0749,E1 11.3456,E2 302.332} C_DIS
LIN {X -114.0897,Y 75.0621,Z 165,A 146.5538,B 11.4811,C 0.0704,E1 11.3485,E2 304.2243} C_DIS
LIN {X -111.6134,Y 78.6971,Z 165,A 144.7074,B 11.4811,C 0.0659,E1 11.3514,E2 306.0688} C_DIS
LIN {X -109.4608,Y 81.6648,Z 165,A 143.1146,B 11.4811,C 0.0634,E1 11.3541,E2 307.6665} C_DIS
LIN {X -106.6184,Y 85.3431,Z 165,A 141.1992,B 11.4811,C 0.0581,E1 11.3574,E2 309.5755} C_DIS
LIN {X -104.1542,Y 88.3329,Z 165,A 139.5175,B 11.4811,C 0.0555,E1 11.3604,E2 311.2622} C_DIS
LIN {X -101.0454,Y 91.8729,Z 165,A 137.5448,B 11.4812,C 0.051,E1 11.364,E2 313.2323} C_DIS
LIN {X -97.9679,Y 95.1479,Z 165,A 135.6478,B 11.4812,C 0.0472,E1 11.3677,E2 315.1287} C_DIS
LIN {X -94.1213,Y 98.9543,Z 165,A 133.025,B 11.4812,C 0.0501,E1 11.373,E2 317.7914} C_DIS
LIN {X -91.3311,Y 101.5357,Z 165,A 131.7655,B 11.4812,C 0.0395,E1 11.3756,E2 319.0089} C_DIS
LIN {X -88.1423,Y 104.3162,Z 165,A 129.3788,B 11.4812,C 0.0495,E1 11.3808,E2 321.4672} C_DIS
LIN {X -84.221,Y 107.5064,Z 165,A 127.6127,B 11.4812,C 0.0377,E1 11.3846,E2 323.1887} C_DIS
LIN {X -79.6289,Y 110.9508,Z 165,A 125.3286,B 11.4812,C 0.0307,E1 11.3897,E2 325.4555} C_DIS
LIN {X -75.9187,Y 113.5216,Z 165,A 123.1585,B 11.4812,C 0.0336,E1 11.3947,E2 327.6569} C_DIS
LIN {X -72.7877,Y 115.554,Z 165,A 121.9624,B 11.4813,C 0.0228,E1 11.3975,E2 328.8071} C_DIS
LIN {X -70.1691,Y 117.163,Z 165,A 120.5942,B 11.4813,C 0.0225,E1 11.4007,E2 330.1836} C_DIS
LIN {X -66.6518,Y 119.199,Z 165,A 118.8421,B 11.4813,C 0.021,E1 11.405,E2 331.9398} C_DIS
LIN {X -63.0886,Y 121.1209,Z 165,A 116.9379,B 11.4813,C 0.0232,E1 11.4098,E2 333.8671} C_DIS
LIN {X -60.1775,Y 122.5927,Z 165,A 115.868,B 11.4813,C 0.0146,E1 11.4124,E2 334.8998} C_DIS
LIN {X -57.1229,Y 124.0454,Z 165,A 114.4136,B 11.4813,C 0.0136,E1 11.416,E2 336.3573} C_DIS
LIN {X -54.0854,Y 125.3995,Z 165,A 112.6621,B 11.4813,C 0.02,E1 11.4206,E2 338.1505} C_DIS
LIN {X -50.6557,Y 126.8245,Z 165,A 111.4789,B 11.4813,C 0.0096,E1 11.4236,E2 339.2873} C_DIS
LIN {X -47.3749,Y 128.0867,Z 165,A 109.9902,B 11.4813,C 0.0083,E1 11.4275,E2 340.7766} C_DIS
LIN {X -41.7955,Y 130.0134,Z 165,A 107.721,B 11.4813,C 0.001,E1 11.4334,E2 343.0187} C_DIS
LIN {X -37.9909,Y 131.176,Z 165,A 105.7015,B 11.4813,C 0.0077,E1 11.4389,E2 345.0794} C_DIS
LIN {X -33.7406,Y 132.3325,Z 165,A 103.9251,B 11.4813,C 0.0045,E1 11.4437,E2 346.8458} C_DIS
LIN {X -30.2697,Y 133.1694,Z 165,A 102.4429,B 11.4813,C 0.0031,E1 11.4477,E2 348.325} C_DIS
LIN {X -26.3272,Y 134.0063,Z 165,A 100.6138,B 11.4813,C 0.0052,E1 11.4527,E2 350.1698} C_DIS
LIN {X -22.1647,Y 134.7559,Z 165,A 98.9497,B 11.4813,C 0.0016,E1 11.4573,E2 351.8194} C_DIS
LIN {X -18.0886,Y 135.3635,Z 165,A 97.1764,B 11.4813,C 0.0019,E1 11.4622,E2 353.597} C_DIS
LIN {X -13.8493,Y 135.8644,Z 165,A 95.5078,B 11.4813,C -0.0017,E1 11.4668,E2 355.2499} C_DIS
LIN {X -9.6422,Y 136.2259,Z 165,A 93.6085,B 11.4813,C 0.0008,E1 11.4721,E2 357.1635} C_DIS
LIN {X -5.4314,Y 136.4584,Z 165,A 91.7554,B 11.4813,C 0.0025,E1 11.4773,E2 359.0258} C_DIS
LIN {X 0.4879,Y 136.5659,Z 165,A 89.5113,B 11.4813,C -0.0035,E1 11.4835,E2 361.2398} C_DIS
LIN {X 3.8498,Y 136.5122,Z 165,A 87.9997,B 11.4813,C -0.001,E1 11.4877,E2 362.763} C_DIS
LIN {X 10.1517,Y 136.1887,Z 165,A 85.2458,B 11.4813,C 0.0019,E1 11.4955,E2 365.5287} C_DIS
LIN {X 14.7005,Y 135.7728,Z 165,A 83.4516,B 11.4813,C -0.0007,E1 11.5004,E2 367.3074} C_DIS
LIN {X 18.6321,Y 135.2911,Z 165,A 81.7667,B 11.4813,C 0.0005,E1 11.5051,E2 368.9947} C_DIS
LIN {X 24.2529,Y 134.3956,Z 165,A 79.4901,B 11.4813,C -0.0013,E1 11.5113,E2 371.2571} C_DIS
LIN {X 27.2509,Y 133.8197,Z 165,A 78.1341,B 11.4813,C 0.0012,E1 11.515,E2 372.6218} C_DIS
LIN {X 30.7145,Y 133.0678,Z 165,A 76.6444,B 11.4813,C 0.0022,E1 11.5191,E2 374.1116} C_DIS
LIN {X 34.3612,Y 132.175,Z 165,A 74.9407,B 11.4813,C 0.0065,E1 11.5238,E2 375.8306} C_DIS
LIN {X 38.2529,Y 131.0993,Z 165,A 73.3462,B 11.4813,C 0.0052,E1 11.528,E2 377.4127} C_DIS
LIN {X 41.803,Y 130.011,Z 165,A 71.8132,B 11.4813,C 0.0059,E1 11.5321,E2 378.9425} C_DIS
LIN {X 45.8607,Y 128.6363,Z 165,A 70.1895,B 11.4813,C 0.0031,E1 11.5363,E2 380.5449} C_DIS
LIN {X 49.1259,Y 127.4247,Z 165,A 67.8276,B 11.4813,C 0.0273,E1 11.5428,E2 383.0157} C_DIS
LIN {X 54.531,Y 125.2068,Z 165,A 66.1615,B 11.4813,C 0.0102,E1 11.5468,E2 384.587} C_DIS
LIN {X 57.412,Y 123.9117,Z 165,A 64.8507,B 11.4813,C 0.0114,E1 11.5501,E2 385.896} C_DIS
LIN {X 60.5558,Y 122.4061,Z 165,A 63.3663,B 11.4813,C 0.0137,E1 11.5538,E2 387.3831} C_DIS
LIN {X 63.8406,Y 120.726,Z 165,A 61.8076,B 11.4813,C 0.016,E1 11.5577,E2 388.9433} C_DIS
LIN {X 67.7518,Y 118.5769,Z 165,A 59.8953,B 11.4813,C 0.0197,E1 11.5624,E2 390.8607} C_DIS
LIN {X 71.432,Y 116.3969,Z 165,A 58.1214,B 11.4813,C 0.0218,E1 11.5666,E2 392.6323} C_DIS
LIN {X 75.2596,Y 113.9597,Z 165,A 56.2618,B 11.4813,C 0.0236,E1 11.571,E2 394.4869} C_DIS
LIN {X 78.834,Y 111.5169,Z 165,A 54.3835,B 11.4813,C 0.0281,E1 11.5753,E2 396.3732} C_DIS
LIN {X 82.1532,Y 109.0947,Z 165,A 52.822,B 11.4813,C 0.0268,E1 11.5788,E2 397.9153} C_DIS
LIN {X 88.2168,Y 104.253,Z 165,A 49.5814,B 11.4813,C 0.0323,E1 11.5858,E2 401.1551} C_DIS
LIN {X 91.2687,Y 101.5915,Z 165,A 47.7877,B 11.4813,C 0.0381,E1 11.5896,E2 402.961} C_DIS
LIN {X 94.3927,Y 98.6955,Z 165,A 46.2242,B 11.4813,C 0.0357,E1 11.5927,E2 404.4977} C_DIS
LIN {X 96.8646,Y 96.2706,Z 165,A 44.5779,B 11.4813,C 0.0437,E1 11.596,E2 406.1684} C_DIS
LIN {X 99.8402,Y 93.1812,Z 165,A 42.5951,B 11.4813,C 0.0524,E1 11.5999,E2 408.1743} C_DIS
LIN {X 102.0832,Y 90.719,Z 165,A 41.4787,B 11.4813,C 0.0479,E1 11.6019,E2 409.2571} C_DIS
LIN {X 104.7968,Y 87.5699,Z 165,A 39.6933,B 11.4813,C 0.0529,E1 11.6051,E2 411.0485} C_DIS
LIN {X 107.641,Y 84.0497,Z 165,A 37.778,B 11.4812,C 0.0576,E1 11.6085,E2 412.9668} C_DIS
LIN {X 110.3557,Y 80.4521,Z 165,A 35.9069,B 11.4812,C 0.0615,E1 11.6116,E2 414.8365} C_DIS
LIN {X 112.9722,Y 76.734,Z 165,A 34.0357,B 11.4812,C 0.065,E1 11.6145,E2 416.7044} C_DIS
LIN {X 115.4698,Y 72.9213,Z 165,A 32.1947,B 11.4812,C 0.0678,E1 11.6173,E2 418.5379} C_DIS
LIN {X 117.5668,Y 69.4909,Z 165,A 30.4886,B 11.4812,C 0.0725,E1 11.6198,E2 420.2475} C_DIS
LIN {X 120.0007,Y 65.1972,Z 165,A 28.4893,B 11.4811,C 0.0758,E1 11.6225,E2 422.2394} C_DIS
LIN {X 121.61,Y 62.1393,Z 165,A 27.016,B 11.4811,C 0.0802,E1 11.6244,E2 423.7166} C_DIS
LIN {X 123.2059,Y 58.9115,Z 165,A 25.5538,B 11.4811,C 0.0828,E1 11.6261,E2 425.1739} C_DIS
LIN {X 124.7413,Y 55.5867,Z 165,A 24.0021,B 11.481,C 0.0873,E1 11.6279,E2 426.7287} C_DIS
LIN {X 126.3476,Y 51.8375,Z 165,A 22.4184,B 11.481,C 0.0884,E1 11.6296,E2 428.2981} C_DIS
LIN {X 127.5406,Y 48.8277,Z 165,A 20.7808,B 11.4809,C 0.0998,E1 11.6313,E2 429.9712} C_DIS
LIN {X 129.1035,Y 44.5266,Z 165,A 19.1837,B 11.4809,C 0.0962,E1 11.6328,E2 431.53} C_DIS
LIN {X 130.1205,Y 41.4601,Z 165,A 17.8161,B 11.4809,C 0.1003,E1 11.634,E2 432.9003} C_DIS
LIN {X 131.2694,Y 37.672,Z 165,A 16.1978,B 11.4809,C 0.1038,E1 11.6352,E2 434.5149} C_DIS
LIN {X 131.9315,Y 35.276,Z 165,A 15.1426,B 11.4809,C 0.107,E1 11.636,E2 435.5725} C_DIS
LIN {X 132.7864,Y 31.9075,Z 165,A 13.7058,B 11.4809,C 0.1106,E1 11.637,E2 437.008} C_DIS
LIN {X 133.6313,Y 28.1682,Z 165,A 12.1613,B 11.4808,C 0.1134,E1 11.6379,E2 438.5462} C_DIS
LIN {X 134.1713,Y 25.4641,Z 165,A 10.9907,B 11.4808,C 0.1171,E1 11.6385,E2 439.7194} C_DIS
LIN {X 134.8201,Y 21.7799,Z 165,A 9.4507,B 11.4807,C 0.1209,E1 11.6392,E2 441.2573} C_DIS
LIN {X 135.3726,Y 18.0186,Z 165,A 7.7639,B 11.4807,C 0.1281,E1 11.6399,E2 442.9571} C_DIS
LIN {X 135.942,Y 13.0438,Z 165,A 5.7701,B 11.4806,C 0.1312,E1 11.6405,E2 444.9396} C_DIS
LIN {X 136.2704,Y 9.0078,Z 165,A 3.6768,B 11.4804,C 0.1471,E1 11.6409,E2 447.0836} C_DIS
LIN {X 136.4728,Y 5.0635,Z 165,A 2.4642,B 11.4804,C 0.1397,E1 11.6411,E2 448.2428} C_DIS
LIN {X 136.5589,Y -1.5919,Z 165,A -0.2242,B 11.4804,C 0.1451,E1 11.6411,E2 450.9213} C_DIS
LIN {X 136.1746,Y -10.3443,Z 165,A -4.1965,B 11.4802,C 0.1642,E1 11.6405,E2 454.9346} C_DIS
LIN {X 135.8884,Y -13.6017,Z 165,A -5.1873,B 11.4802,C 0.1576,E1 11.6403,E2 455.8795} C_DIS
LIN {X 135.5868,Y -16.3278,Z 165,A -6.4324,B 11.4802,C 0.1636,E1 11.6399,E2 457.1375} C_DIS
LIN {X 135.122,Y -19.8152,Z 165,A -7.8473,B 11.4802,C 0.1662,E1 11.6393,E2 458.5466} C_DIS
LIN {X 134.3846,Y -24.3142,Z 165,A -9.8989,B 11.48,C 0.1757,E1 11.6384,E2 460.6176} C_DIS
LIN {X 133.7544,Y -27.5717,Z 165,A -11.2143,B 11.48,C 0.1776,E1 11.6376,E2 461.925} C_DIS
LIN {X 132.7721,Y -31.9667,Z 165,A -13.0586,B 11.48,C 0.1818,E1 11.6365,E2 463.7658} C_DIS
LIN {X 131.8752,Y -35.4869,Z 165,A -14.4747,B 11.4799,C 0.1832,E1 11.6355,E2 465.1701} C_DIS
LIN {X 131.0153,Y -38.5397,Z 165,A -15.7845,B 11.4799,C 0.1864,E1 11.6345,E2 466.4789} C_DIS
LIN {X 130.0802,Y -41.5863,Z 165,A -17.1482,B 11.4798,C 0.191,E1 11.6333,E2 467.8474} C_DIS
LIN {X 128.9481,Y -44.9748,Z 165,A -18.6515,B 11.4797,C 0.1954,E1 11.632,E2 469.3531} C_DIS
LIN {X 126.9261,Y -50.4036,Z 165,A -20.9561,B 11.4797,C 0.1987,E1 11.6297,E2 471.6448} C_DIS
LIN {X 125.0459,Y -54.9032,Z 165,A -23.065,B 11.4795,C 0.2061,E1 11.6274,E2 473.7639} C_DIS
LIN {X 123.3597,Y -58.5894,Z 165,A -25.3333,B 11.4791,C 0.2263,E1 11.6246,E2 476.1048} C_DIS
LIN {X 121.0927,Y -63.1423,Z 165,A -26.6513,B 11.4794,C 0.2095,E1 11.6231,E2 477.3236} C_DIS
LIN {X 119.5593,Y -66.0031,Z 165,A -28.2714,B 11.4792,C 0.2203,E1 11.6208,E2 478.9778} C_DIS
LIN {X 117.2716,Y -69.987,Z 165,A -30.1191,B 11.4792,C 0.2231,E1 11.6182,E2 480.8177} C_DIS
LIN {X 115.0696,Y -73.5513,Z 165,A -31.9137,B 11.4791,C 0.2286,E1 11.6156,E2 482.6189} C_DIS
LIN {X 112.4641,Y -77.4769,Z 165,A -33.8302,B 11.4791,C 0.2319,E1 11.6126,E2 484.5301} C_DIS
LIN {X 110.0196,Y -80.9103,Z 165,A -35.8293,B 11.4788,C 0.2426,E1 11.6093,E2 486.5602} C_DIS
LIN {X 107.9616,Y -83.6366,Z 165,A -36.7931,B 11.479,C 0.2332,E1 11.6077,E2 487.4668} C_DIS
LIN {X 104.0142,Y -88.4976,Z 165,A -39.5814,B 11.4788,C 0.2438,E1 11.6027,E2 490.2784} C_DIS
LIN {X 99.9626,Y -93.0497,Z 165,A -41.8746,B 11.4788,C 0.2425,E1 11.5985,E2 492.5413} C_DIS
LIN {X 97.8557,Y -95.2638,Z 165,A -43.4351,B 11.4786,C 0.2529,E1 11.5954,E2 494.1382} C_DIS
LIN {X 94.8192,Y -98.2861,Z 165,A -45.1829,B 11.4786,C 0.2554,E1 11.5919,E2 495.8817} C_DIS
LIN {X 91.9093,Y -101.0123,Z 165,A -46.8688,B 11.4784,C 0.2592,E1 11.5885,E2 497.571} C_DIS
LIN {X 88.5667,Y -103.9555,Z 165,A -48.7298,B 11.4784,C 0.2628,E1 11.5845,E2 499.4331} C_DIS
LIN {X 85.1393,Y -106.7806,Z 165,A -50.5386,B 11.4784,C 0.265,E1 11.5806,E2 501.237} C_DIS
LIN {X 81.8219,Y -109.3438,Z 165,A -52.3408,B 11.4782,C 0.2695,E1 11.5766,E2 503.0464} C_DIS
LIN {X 78.1962,Y -111.9652,Z 165,A -54.1961,B 11.4782,C 0.2723,E1 11.5724,E2 504.9008} C_DIS
LIN {X 72.7641,Y -115.569,Z 165,A -56.8452,B 11.4781,C 0.2747,E1 11.5662,E2 507.5418} C_DIS
LIN {X 69.0518,Y -117.8247,Z 165,A -58.6698,B 11.4781,C 0.2777,E1 11.5618,E2 509.3685} C_DIS
LIN {X 65.0809,Y -120.0641,Z 165,A -60.605,B 11.4779,C 0.2813,E1 11.5571,E2 511.3082} C_DIS
LIN {X 60.3267,Y -122.5191,Z 165,A -62.8985,B 11.4779,C 0.2858,E1 11.5514,E2 513.6098} C_DIS
LIN {X 55.6013,Y -124.7348,Z 165,A -64.8403,B 11.4779,C 0.2822,E1 11.5465,E2 515.5224} C_DIS
LIN {X 52.7334,Y -125.974,Z 165,A -66.2921,B 11.4778,C 0.2876,E1 11.5427,E2 516.9931} C_DIS
LIN {X 49.0923,Y -127.4378,Z 165,A -67.8153,B 11.4778,C 0.2863,E1 11.5388,E2 518.5022} C_DIS
LIN {X 46.1191,Y -128.5432,Z 165,A -69.171,B 11.4778,C 0.2885,E1 11.5352,E2 519.8621} C_DIS
LIN {X 42.8689,Y -129.6635,Z 165,A -70.6326,B 11.4777,C 0.2905,E1 11.5314,E2 521.3272} C_DIS
LIN {X 39.6749,Y -130.6763,Z 165,A -72.0747,B 11.4777,C 0.2929,E1 11.5275,E2 522.775} C_DIS
LIN {X 35.3252,Y -131.9184,Z 165,A -73.907,B 11.4777,C 0.2929,E1 11.5226,E2 524.6005} C_DIS
LIN {X 31.8886,Y -132.791,Z 165,A -75.4065,B 11.4776,C 0.2945,E1 11.5185,E2 526.1025} C_DIS
LIN {X 27.8814,Y -133.6914,Z 165,A -77.3439,B 11.4774,C 0.3013,E1 11.5132,E2 528.0681} C_DIS
LIN {X 22.7376,Y -134.6603,Z 165,A -79.3089,B 11.4775,C 0.2968,E1 11.5078,E2 530.0055} C_DIS
LIN {X 18.6388,Y -135.2901,Z 165,A -81.1285,B 11.4775,C 0.2998,E1 11.5028,E2 531.8363} C_DIS
LIN {X 14.5487,Y -135.7892,Z 165,A -82.768,B 11.4775,C 0.2984,E1 11.4983,E2 533.4655} C_DIS
LIN {X 9.0605,Y -136.2671,Z 165,A -84.9833,B 11.4775,C 0.2968,E1 11.4921,E2 535.6702} C_DIS
LIN {X 1.8395,Y -136.5548,Z 165,A -89.0112,B 11.4769,C 0.3222,E1 11.4805,E2 539.8235} C_DIS
LIN {X 1.8395,Y -136.5548,Z 165,A -89.0112,B 11.4769,C 0.3222,E1 11.4805,E2 539.8235} C_DIS
Enddeposition()
LIN {X 0.9794,Y -137.4792,Z 165,A -87.9528,B 11.3942,C 0.2979,E1 11.4005,E2 538.6477} C_DIS
Startdeposition()
$VEL.CP = VEL_PRINT
LIN {X 6.2353,Y -137.3447,Z 165,A -85.4869,B 11.3943,C 0.2904,E1 11.4075,E2 536.1456} C_DIS
LIN {X 13.452,Y -136.8251,Z 165,A -82.6419,B 11.3943,C 0.2937,E1 11.4153,E2 533.3209} C_DIS
LIN {X 17.6991,Y -136.3405,Z 165,A -80.7462,B 11.3943,C 0.2899,E1 11.4206,E2 531.4095} C_DIS
LIN {X 21.5093,Y -135.7922,Z 165,A -79.1565,B 11.3943,C 0.2893,E1 11.425,E2 529.8206} C_DIS
LIN {X 28.7982,Y -134.4345,Z 165,A -76.1138,B 11.3943,C 0.2885,E1 11.4333,E2 526.7821} C_DIS
LIN {X 32.2499,Y -133.6483,Z 165,A -74.6256,B 11.3944,C 0.2869,E1 11.4374,E2 525.2912} C_DIS
LIN {X 35.7037,Y -132.7676,Z 165,A -73.1051,B 11.3944,C 0.2847,E1 11.4415,E2 523.7651} C_DIS
LIN {X 39.8975,Y -131.5683,Z 165,A -71.3015,B 11.3945,C 0.2834,E1 11.4463,E2 521.9619} C_DIS
LIN {X 42.7944,Y -130.656,Z 165,A -70.1329,B 11.3945,C 0.2846,E1 11.4494,E2 520.8049} C_DIS
LIN {X 46.3538,Y -129.4345,Z 165,A -68.4192,B 11.3946,C 0.279,E1 11.454,E2 519.0712} C_DIS
LIN {X 50.0019,Y -128.0692,Z 165,A -66.877,B 11.3946,C 0.2793,E1 11.458,E2 517.5381} C_DIS
LIN {X 53.7754,Y -126.5337,Z 165,A -65.0688,B 11.3947,C 0.2742,E1 11.4627,E2 515.7143} C_DIS
LIN {X 58.002,Y -124.6505,Z 165,A -62.6258,B 11.3951,C 0.2578,E1 11.4691,E2 513.2031} C_DIS
LIN {X 62.8394,Y -122.2838,Z 165,A -61.4219,B 11.3945,C 0.2825,E1 11.4717,E2 512.1311} C_DIS
LIN {X 68.1399,Y -119.4125,Z 165,A -58.7309,B 11.3947,C 0.274,E1 11.4784,E2 509.4152} C_DIS
LIN {X 74.2091,Y -115.7386,Z 165,A -55.5976,B 11.395,C 0.2644,E1 11.4859,E2 506.2567} C_DIS
LIN {X 77.4902,Y -113.5685,Z 165,A -53.8939,B 11.395,C 0.2598,E1 11.4899,E2 504.5431} C_DIS
LIN {X 81.1637,Y -110.9727,Z 165,A -52.0237,B 11.3951,C 0.2565,E1 11.4941,E2 502.6716} C_DIS
LIN {X 84.835,Y -108.1916,Z 165,A -50.1644,B 11.3951,C 0.2544,E1 11.4982,E2 500.818} C_DIS
LIN {X 88.2366,Y -105.4359,Z 165,A -48.3385,B 11.3953,C 0.2508,E1 11.5022,E2 498.99} C_DIS
LIN {X 91.6445,Y -102.4875,Z 165,A -46.4943,B 11.3953,C 0.2479,E1 11.506,E2 497.1482} C_DIS
LIN {X 94.7944,Y -99.5816,Z 165,A -44.6978,B 11.3954,C 0.2439,E1 11.5097,E2 495.3484} C_DIS
LIN {X 97.9496,Y -96.4798,Z 165,A -42.9004,B 11.3954,C 0.2411,E1 11.5132,E2 493.5549} C_DIS
LIN {X 100.9526,Y -93.3334,Z 165,A -41.2305,B 11.3954,C 0.2411,E1 11.5164,E2 491.9014} C_DIS
LIN {X 103.053,Y -91.008,Z 165,A -39.8103,B 11.3956,C 0.2349,E1 11.5191,E2 490.4651} C_DIS
LIN {X 104.9832,Y -88.7753,Z 165,A -38.457,B 11.3957,C 0.2286,E1 11.5215,E2 489.0946} C_DIS
LIN {X 108.3284,Y -84.6609,Z 165,A -36.6508,B 11.3957,C 0.2346,E1 11.5246,E2 487.3377} C_DIS
LIN {X 111.5022,Y -80.4347,Z 165,A -34.1587,B 11.3959,C 0.2212,E1 11.5288,E2 484.8061} C_DIS
LIN {X 114.136,Y -76.652,Z 165,A -32.2878,B 11.3959,C 0.2178,E1 11.5317,E2 482.9394} C_DIS
LIN {X 116.5577,Y -72.9164,Z 165,A -30.6078,B 11.3959,C 0.2179,E1 11.5342,E2 481.2797} C_DIS
LIN {X 118.5918,Y -69.5585,Z 165,A -28.9036,B 11.3961,C 0.2118,E1 11.5367,E2 479.5649} C_DIS
LIN {X 120.7384,Y -65.762,Z 165,A -27.0709,B 11.3961,C 0.2066,E1 11.5392,E2 477.7281} C_DIS
LIN {X 122.6837,Y -62.0538,Z 165,A -25.0039,B 11.3964,C 0.1928,E1 11.5419,E2 475.6178} C_DIS
LIN {X 124.5068,Y -58.3126,Z 165,A -23.7716,B 11.3962,C 0.2023,E1 11.5433,E2 474.4479} C_DIS
LIN {X 126.7511,Y -53.2551,Z 165,A -21.4382,B 11.3963,C 0.1952,E1 11.5459,E2 472.1084} C_DIS
LIN {X 129.1391,Y -47.1731,Z 165,A -18.653,B 11.3965,C 0.1859,E1 11.5487,E2 469.3121} C_DIS
LIN {X 130.3597,Y -43.6842,Z 165,A -17.2403,B 11.3965,C 0.1851,E1 11.5499,E2 467.914} C_DIS
LIN {X 131.3848,Y -40.497,Z 165,A -15.8139,B 11.3965,C 0.1802,E1 11.5511,E2 466.4819} C_DIS
LIN {X 132.2775,Y -37.4806,Z 165,A -14.5286,B 11.3966,C 0.1772,E1 11.5521,E2 465.1985} C_DIS
LIN {X 133.1238,Y -34.3549,Z 165,A -13.2453,B 11.3966,C 0.1752,E1 11.553,E2 463.9221} C_DIS
LIN {X 133.9808,Y -30.8401,Z 165,A -11.7241,B 11.3967,C 0.1705,E1 11.554,E2 462.3975} C_DIS
LIN {X 134.7101,Y -27.4793,Z 165,A -9.7047,B 11.397,C 0.1497,E1 11.5552,E2 460.3013} C_DIS
LIN {X 135.642,Y -22.4331,Z 165,A -7.6309,B 11.397,C 0.1453,E1 11.5561,E2 458.2335} C_DIS
LIN {X 136.3596,Y -17.5529,Z 165,A -6.0845,B 11.397,C 0.1537,E1 11.5567,E2 456.7501} C_DIS
LIN {X 137.0252,Y -11.2338,Z 165,A -3.5415,B 11.397,C 0.1489,E1 11.5574,E2 454.2175} C_DIS
LIN {X 137.4256,Y -4.0309,Z 165,A -0.6033,B 11.3971,C 0.142,E1 11.5578,E2 451.285} C_DIS
LIN {X 137.481,Y -1.1227,Z 165,A 1.405,B 11.3974,C 0.1158,E1 11.5578,E2 449.1737} C_DIS
LIN {X 137.3932,Y 5.0222,Z 165,A 3.5641,B 11.3974,C 0.1197,E1 11.5576,E2 447.0635} C_DIS
LIN {X 137.1744,Y 9.256,Z 165,A 5.0849,B 11.3974,C 0.1215,E1 11.5573,E2 445.5724} C_DIS
LIN {X 136.3848,Y 17.3612,Z 165,A 8.4003,B 11.3974,C 0.1138,E1 11.5563,E2 442.2636} C_DIS
LIN {X 135.6637,Y 22.3025,Z 165,A 10.334,B 11.3974,C 0.1119,E1 11.5555,E2 440.3465} C_DIS
LIN {X 135.0126,Y 25.9526,Z 165,A 11.758,B 11.3974,C 0.1109,E1 11.5548,E2 438.9364} C_DIS
LIN {X 134.1727,Y 30.0002,Z 165,A 13.6112,B 11.3975,C 0.1023,E1 11.5537,E2 437.0651} C_DIS
LIN {X 133.4228,Y 33.1771,Z 165,A 14.9868,B 11.3975,C 0.098,E1 11.5528,E2 435.6864} C_DIS
LIN {X 132.3316,Y 37.2872,Z 165,A 16.6124,B 11.3975,C 0.0971,E1 11.5516,E2 434.0777} C_DIS
LIN {X 131.213,Y 41.0573,Z 165,A 18.2725,B 11.3976,C 0.0919,E1 11.5502,E2 432.4136} C_DIS
LIN {X 129.9687,Y 44.8338,Z 165,A 19.8627,B 11.3976,C 0.0892,E1 11.5488,E2 430.8303} C_DIS
LIN {X 127.3777,Y 51.7391,Z 165,A 22.9175,B 11.3977,C 0.0814,E1 11.5458,E2 427.7755} C_DIS
LIN {X 125.763,Y 55.5513,Z 165,A 24.6661,B 11.3977,C 0.0761,E1 11.5438,E2 426.0227} C_DIS
LIN {X 123.7414,Y 59.9203,Z 165,A 26.7089,B 11.3977,C 0.0699,E1 11.5414,E2 423.9738} C_DIS
LIN {X 121.8386,Y 63.6967,Z 165,A 28.3024,B 11.3977,C 0.0699,E1 11.5393,E2 422.4002} C_DIS
LIN {X 118.287,Y 70.0765,Z 165,A 31.4535,B 11.3978,C 0.0593,E1 11.535,E2 419.2336} C_DIS
LIN {X 115.997,Y 73.8055,Z 165,A 33.2148,B 11.3978,C 0.0566,E1 11.5324,E2 417.479} C_DIS
LIN {X 113.6405,Y 77.3847,Z 165,A 34.9025,B 11.3978,C 0.0549,E1 11.5298,E2 415.8025} C_DIS
LIN {X 111.2798,Y 80.7415,Z 165,A 36.6534,B 11.3978,C 0.0498,E1 11.5269,E2 414.0455} C_DIS
LIN {X 108.6526,Y 84.2438,Z 165,A 38.4602,B 11.3979,C 0.0461,E1 11.5239,E2 412.2399} C_DIS
LIN {X 105.9352,Y 87.6364,Z 165,A 40.2691,B 11.3979,C 0.0421,E1 11.5207,E2 410.4305} C_DIS
LIN {X 102.9394,Y 91.1366,Z 165,A 42.9617,B 11.3979,C 0.0169,E1 11.5155,E2 407.6394} C_DIS
LIN {X 98.4943,Y 95.9241,Z 165,A 44.9004,B 11.3979,C 0.0325,E1 11.512,E2 405.7986} C_DIS
LIN {X 95.9978,Y 98.4223,Z 165,A 46.4933,B 11.3979,C 0.0263,E1 11.5088,E2 404.1899} C_DIS
LIN {X 92.0344,Y 102.1383,Z 165,A 48.621,B 11.3979,C 0.0256,E1 11.5044,E2 402.0785} C_DIS
LIN {X 88.9092,Y 104.8694,Z 165,A 50.2532,B 11.3979,C 0.0249,E1 11.501,E2 400.4579} C_DIS
LIN {X 84.4066,Y 108.5264,Z 165,A 52.707,B 11.3979,C 0.0197,E1 11.4956,E2 397.9989} C_DIS
LIN {X 80.7384,Y 111.2821,Z 165,A 54.6109,B 11.3979,C 0.0166,E1 11.4913,E2 396.0955} C_DIS
LIN {X 76.9165,Y 113.9574,Z 165,A 56.4989,B 11.3979,C 0.015,E1 11.487,E2 394.2142} C_DIS
LIN {X 73.1352,Y 116.4205,Z 165,A 58.3945,B 11.3979,C 0.0117,E1 11.4825,E2 392.3163} C_DIS
LIN {X 69.2674,Y 118.7629,Z 165,A 60.2838,B 11.3979,C 0.0088,E1 11.478,E2 390.4262} C_DIS
LIN {X 65.3795,Y 120.9464,Z 165,A 62.1355,B 11.3979,C 0.0065,E1 11.4735,E2 388.5752} C_DIS
LIN {X 61.3057,Y 123.0599,Z 165,A 63.8934,B 11.3979,C 0.008,E1 11.4691,E2 386.8363} C_DIS
LIN {X 58.0224,Y 124.641,Z 165,A 65.4473,B 11.3979,C 0.0053,E1 11.4652,E2 385.278} C_DIS
LIN {X 55.5154,Y 125.779,Z 165,A 66.5868,B 11.3979,C 0.0042,E1 11.4623,E2 384.1395} C_DIS
LIN {X 50.5632,Y 127.851,Z 165,A 68.9687,B 11.3979,C -0.0019,E1 11.4561,E2 381.7397} C_DIS
LIN {X 47.1626,Y 129.1429,Z 165,A 70.2974,B 11.3979,C 0.0014,E1 11.4527,E2 380.4344} C_DIS
LIN {X 43.6842,Y 130.3597,Z 165,A 71.8242,B 11.3979,C 0.0002,E1 11.4487,E2 378.9088} C_DIS
LIN {X 40.3372,Y 131.4337,Z 165,A 73.1949,B 11.3979,C 0.0014,E1 11.445,E2 377.55} C_DIS
LIN {X 37.1101,Y 132.3811,Z 165,A 74.7834,B 11.3979,C -0.0044,E1 11.4407,E2 375.9386} C_DIS
LIN {X 32.4692,Y 133.5954,Z 165,A 76.6765,B 11.3979,C -0.0031,E1 11.4356,E2 374.059} C_DIS
LIN {X 28.9701,Y 134.3974,Z 165,A 78.1665,B 11.3979,C -0.0038,E1 11.4316,E2 372.5701} C_DIS
LIN {X 25.3902,Y 135.1202,Z 165,A 80.7151,B 11.3979,C -0.0304,E1 11.4242,E2 369.8936} C_DIS
LIN {X 18.2329,Y 136.2705,Z 165,A 82.787,B 11.3979,C -0.0076,E1 11.4188,E2 367.9415} C_DIS
LIN {X 14.0356,Y 136.7678,Z 165,A 85.0486,B 11.3979,C -0.0205,E1 11.4124,E2 365.6183} C_DIS
LIN {X 9.179,Y 137.1797,Z 165,A 87.25,B 11.3979,C -0.0251,E1 11.4062,E2 363.3965} C_DIS
LIN {X 3.4712,Y 137.4412,Z 165,A 88.8531,B 11.3979,C -0.0059,E1 11.402,E2 361.8912} C_DIS
LIN {X -1.3822,Y 137.4791,Z 165,A 91.1559,B 11.3979,C -0.0127,E1 11.3954,E2 359.5548} C_DIS
LIN {X -5.0262,Y 137.393,Z 165,A 92.8753,B 11.3979,C -0.0173,E1 11.3906,E2 357.8111} C_DIS
LIN {X -9.2814,Y 137.1728,Z 165,A 94.3162,B 11.3979,C -0.0087,E1 11.3867,E2 356.4129} C_DIS
LIN {X -12.436,Y 136.9227,Z 165,A 96.0219,B 11.3979,C -0.0177,E1 11.3818,E2 354.6599} C_DIS
LIN {X -16.7735,Y 136.4583,Z 165,A 97.4882,B 11.3979,C -0.0084,E1 11.3779,E2 353.2383} C_DIS
LIN {X -20.9511,Y 135.8787,Z 165,A 98.9767,B 11.3979,C -0.0012,E1 11.3738,E2 351.7841} C_DIS
LIN {X -23.9764,Y 135.3778,Z 165,A 100.4337,B 11.3979,C -0.0047,E1 11.3698,E2 350.3058} C_DIS
LIN {X -27.7527,Y 134.6545,Z 165,A 102.1,B 11.3979,C -0.0052,E1 11.3652,E2 348.6327} C_DIS
LIN {X -31.4432,Y 133.8427,Z 165,A 103.689,B 11.3979,C -0.0044,E1 11.3609,E2 347.0431} C_DIS
LIN {X -35.1436,Y 132.917,Z 165,A 105.1209,B 11.3979,C 0.0005,E1 11.357,E2 345.6318} C_DIS
LIN {X -38.5174,Y 131.9785,Z 165,A 106.4963,B 11.3979,C 0.0037,E1 11.3534,E2 344.2677} C_DIS
LIN {X -41.5236,Y 131.0641,Z 165,A 108.5753,B 11.3979,C -0.0132,E1 11.3476,E2 342.0944} C_DIS
LIN {X -46.3504,Y 129.4357,Z 165,A 110.2733,B 11.3979,C -0.001,E1 11.3433,E2 340.4509} C_DIS
LIN {X -50.5552,Y 127.8541,Z 165,A 112.5238,B 11.3979,C -0.0077,E1 11.3373,E2 338.1551} C_DIS
LIN {X -54.8222,Y 126.0812,Z 165,A 113.9221,B 11.3979,C 0.0069,E1 11.3339,E2 336.8238} C_DIS
LIN {X -58.6349,Y 124.3555,Z 165,A 115.7489,B 11.3979,C 0.0073,E1 11.3292,E2 334.9883} C_DIS
LIN {X -65.3297,Y 120.9732,Z 165,A 118.8924,B 11.3979,C 0.0113,E1 11.3214,E2 331.8455} C_DIS
LIN {X -69.2327,Y 118.783,Z 165,A 120.8008,B 11.3979,C 0.0131,E1 11.3168,E2 329.9335} C_DIS
LIN {X -74.2594,Y 115.7064,Z 165,A 124.0364,B 11.3979,C -0.0008,E1 11.309,E2 326.6033} C_DIS
LIN {X -79.6389,Y 112.0723,Z 165,A 125.9821,B 11.3979,C 0.0213,E1 11.3047,E2 324.7549} C_DIS
LIN {X -85.4549,Y 107.7029,Z 165,A 128.7792,B 11.3979,C 0.0321,E1 11.2986,E2 321.9898} C_DIS
LIN {X -90.6074,Y 103.4058,Z 165,A 131.6259,B 11.3979,C 0.0365,E1 11.2925,E2 319.14} C_DIS
LIN {X -95.9229,Y 98.4954,Z 165,A 135.1888,B 11.3979,C 0.0305,E1 11.2851,E2 315.5126} C_DIS
LIN {X -98.5958,Y 95.8192,Z 165,A 136.5837,B 11.3979,C 0.0379,E1 11.2824,E2 314.1419} C_DIS
LIN {X -100.9368,Y 93.3506,Z 165,A 138.4325,B 11.3979,C 0.0314,E1 11.2789,E2 312.2412} C_DIS
LIN {X -104.2278,Y 89.6603,Z 165,A 140.153,B 11.3979,C 0.0437,E1 11.2758,E2 310.5653} C_DIS
LIN {X -107.6376,Y 85.5369,Z 165,A 142.2486,B 11.3979,C 0.0518,E1 11.2721,E2 308.4888} C_DIS
LIN {X -110.4802,Y 81.833,Z 165,A 144.2869,B 11.3979,C 0.0545,E1 11.2687,E2 306.4413} C_DIS
LIN {X -113.1204,Y 78.1432,Z 165,A 146.1673,B 11.3979,C 0.0593,E1 11.2657,E2 304.5643} C_DIS
LIN {X -115.6503,Y 74.3471,Z 165,A 148.0823,B 11.3979,C 0.0638,E1 11.2628,E2 302.6497} C_DIS
LIN {X -118.1024,Y 70.3862,Z 165,A 149.9733,B 11.3978,C 0.0698,E1 11.26,E2 300.7671} C_DIS
LIN {X -120.1299,Y 66.8677,Z 165,A 151.7455,B 11.3978,C 0.0725,E1 11.2576,E2 298.9871} C_DIS
LIN {X -121.7548,Y 63.8562,Z 165,A 153.2293,B 11.3978,C 0.075,E1 11.2556,E2 297.4976} C_DIS
LIN {X -123.9259,Y 59.5342,Z 165,A 155.1028,B 11.3977,C 0.0834,E1 11.2533,E2 295.6441} C_DIS
LIN {X -125.2366,Y 56.7281,Z 165,A 156.4329,B 11.3977,C 0.0861,E1 11.2518,E2 294.3106} C_DIS
LIN {X -126.6887,Y 53.4044,Z 165,A 157.8635,B 11.3977,C 0.092,E1 11.2502,E2 292.8917} C_DIS
LIN {X -128.9473,Y 47.6948,Z 165,A 160.4762,B 11.3976,C 0.0979,E1 11.2476,E2 290.2754} C_DIS
LIN {X -130.4467,Y 43.4228,Z 165,A 162.5642,B 11.3976,C 0.0989,E1 11.2457,E2 288.1646} C_DIS
LIN {X -131.8879,Y 38.8269,Z 165,A 164.2452,B 11.3975,C 0.1116,E1 11.2443,E2 286.5264} C_DIS
LIN {X -132.6175,Y 36.2648,Z 165,A 165.7534,B 11.3975,C 0.1062,E1 11.2432,E2 284.9701} C_DIS
LIN {X -133.5488,Y 32.6625,Z 165,A 167.1916,B 11.3975,C 0.1131,E1 11.2422,E2 283.5477} C_DIS
LIN {X -134.3925,Y 28.993,Z 165,A 168.7086,B 11.3974,C 0.1187,E1 11.2413,E2 282.0389} C_DIS
LIN {X -135.0248,Y 25.889,Z 165,A 170.0724,B 11.3974,C 0.1216,E1 11.2405,E2 280.6712} C_DIS
LIN {X -135.6087,Y 22.6324,Z 165,A 171.5443,B 11.3974,C 0.1236,E1 11.2398,E2 279.1892} C_DIS
LIN {X -136.2124,Y 18.6749,Z 165,A 173.2891,B 11.3973,C 0.1269,E1 11.2391,E2 277.4368} C_DIS
LIN {X -136.7259,Y 14.4247,Z 165,A 175.3376,B 11.3973,C 0.1264,E1 11.2385,E2 275.3572} C_DIS
LIN {X -137.0566,Y 10.8614,Z 165,A 176.6546,B 11.3973,C 0.1346,E1 11.2382,E2 274.0637} C_DIS
LIN {X -137.3193,Y 6.7403,Z 165,A 178.3427,B 11.3971,C 0.1403,E1 11.2379,E2 272.3814} C_DIS
LIN {X -137.4632,Y 2.4301,Z 165,A 179.8803,B 11.3971,C 0.1512,E1 11.2379,E2 270.8781} C_DIS
LIN {X -137.4752,Y -1.7075,Z 165,A -178.1458,B 11.3971,C 0.1509,E1 11.2379,E2 268.8751} C_DIS
LIN {X -137.3869,Y -5.1849,Z 165,A -176.6633,B 11.397,C 0.1545,E1 11.2379,E2 267.3899} C_DIS
LIN {X -137.173,Y -9.2791,Z 165,A -174.8367,B 11.397,C 0.1569,E1 11.2383,E2 265.5504} C_DIS
LIN {X -136.8633,Y -13.0549,Z 165,A -173.3804,B 11.3968,C 0.1642,E1 11.2386,E2 264.1109} C_DIS
LIN {X -136.4733,Y -16.6473,Z 165,A -171.7183,B 11.3968,C 0.1652,E1 11.2392,E2 262.4307} C_DIS
LIN {X -135.8948,Y -20.8466,Z 165,A -170.0507,B 11.3968,C 0.1725,E1 11.2398,E2 260.7773} C_DIS
LIN {X -135.3378,Y -24.1998,Z 165,A -168.6323,B 11.3966,C 0.1765,E1 11.2405,E2 259.36} C_DIS
LIN {X -134.6515,Y -27.7674,Z 165,A -167.0751,B 11.3966,C 0.1799,E1 11.2414,E2 257.7989} C_DIS
LIN {X -133.8828,Y -31.2691,Z 165,A -165.5149,B 11.3966,C 0.1827,E1 11.2423,E2 256.2317} C_DIS
LIN {X -132.9703,Y -34.9438,Z 165,A -163.337,B 11.3966,C 0.174,E1 11.2439,E2 253.9797} C_DIS
LIN {X -131.5929,Y -39.817,Z 165,A -161.481,B 11.3966,C 0.1855,E1 11.2454,E2 252.1577} C_DIS
LIN {X -130.5236,Y -43.1921,Z 165,A -160.2903,B 11.3963,C 0.1959,E1 11.2464,E2 251.0041} C_DIS
LIN {X -128.5451,Y -48.7686,Z 165,A -157.6993,B 11.3963,C 0.1999,E1 11.2489,E2 248.3995} C_DIS
LIN {X -127.1232,Y -52.3641,Z 165,A -156.1225,B 11.3962,C 0.2049,E1 11.2505,E2 246.8283} C_DIS
LIN {X -125.6233,Y -55.8634,Z 165,A -154.5771,B 11.3961,C 0.2101,E1 11.2523,E2 245.2892} C_DIS
LIN {X -124.3235,Y -58.7018,Z 165,A -153.2327,B 11.3961,C 0.2125,E1 11.2539,E2 243.9405} C_DIS
LIN {X -122.7379,Y -61.9475,Z 165,A -151.7638,B 11.396,C 0.2172,E1 11.2557,E2 242.4773} C_DIS
LIN {X -120.9724,Y -65.3311,Z 165,A -150.0591,B 11.396,C 0.2187,E1 11.2579,E2 240.7593} C_DIS
LIN {X -118.7684,Y -69.2579,Z 165,A -148.119,B 11.3959,C 0.222,E1 11.2606,E2 238.8125} C_DIS
LIN {X -116.4786,Y -73.0431,Z 165,A -146.4293,B 11.3957,C 0.23,E1 11.2631,E2 237.1434} C_DIS
LIN {X -113.1373,Y -78.1183,Z 165,A -143.6323,B 11.3957,C 0.23,E1 11.2675,E2 234.3147} C_DIS
LIN {X -110.9488,Y -81.1962,Z 165,A -142.0293,B 11.3957,C 0.2331,E1 11.2701,E2 232.7088} C_DIS
LIN {X -107.9576,Y -85.133,Z 165,A -140.0651,B 11.3955,C 0.2399,E1 11.2734,E2 230.758} C_DIS
LIN {X -105.3497,Y -88.3393,Z 165,A -137.8436,B 11.3957,C 0.2323,E1 11.2775,E2 228.4739} C_DIS
LIN {X -102.1873,Y -91.9797,Z 165,A -136.2806,B 11.3954,C 0.2468,E1 11.2803,E2 226.9688} C_DIS
LIN {X -99.0835,Y -95.3154,Z 165,A -134.3549,B 11.3953,C 0.2501,E1 11.284,E2 225.0405} C_DIS
LIN {X -95.9743,Y -98.4454,Z 165,A -132.4901,B 11.3953,C 0.2531,E1 11.2877,E2 223.1731} C_DIS
LIN {X -92.6397,Y -101.5893,Z 165,A -130.7473,B 11.3951,C 0.2606,E1 11.2913,E2 221.4522} C_DIS
LIN {X -88.1559,Y -105.5033,Z 165,A -127.7972,B 11.3951,C 0.2543,E1 11.2976,E2 218.4432} C_DIS
LIN {X -85.1686,Y -107.9296,Z 165,A -126.624,B 11.3949,C 0.2671,E1 11.3001,E2 217.3253} C_DIS
LIN {X -83.1432,Y -109.4973,Z 165,A -125.3396,B 11.3949,C 0.2638,E1 11.303,E2 216.0136} C_DIS
LIN {X -79.1622,Y -112.4089,Z 165,A -123.3783,B 11.3949,C 0.2693,E1 11.3074,E2 214.0648} C_DIS
LIN {X -75.5912,Y -114.8406,Z 165,A -121.545,B 11.3949,C 0.2713,E1 11.3117,E2 212.2276} C_DIS
LIN {X -72.0182,Y -117.1145,Z 165,A -119.7708,B 11.3948,C 0.2737,E1 11.3159,E2 210.4525} C_DIS
LIN {X -68.5289,Y -119.1904,Z 165,A -118.0074,B 11.3948,C 0.2743,E1 11.3202,E2 208.6803} C_DIS
LIN {X -64.6202,Y -121.3536,Z 165,A -116.163,B 11.3947,C 0.2771,E1 11.3247,E2 206.8381} C_DIS
LIN {X -61.072,Y -123.1752,Z 165,A -114.6031,B 11.3946,C 0.2816,E1 11.3285,E2 205.2913} C_DIS
LIN {X -58.3134,Y -124.5065,Z 165,A -113.2787,B 11.3946,C 0.2819,E1 11.3319,E2 203.9609} C_DIS
LIN {X -53.4668,Y -126.6627,Z 165,A -111.0411,B 11.3946,C 0.2836,E1 11.3376,E2 201.7199} C_DIS
LIN {X -50.1814,Y -127.9994,Z 165,A -109.6378,B 11.3944,C 0.2868,E1 11.3412,E2 200.326} C_DIS
LIN {X -46.7586,Y -129.2886,Z 165,A -108.0602,B 11.3944,C 0.2868,E1 11.3454,E2 198.7415} C_DIS
LIN {X -43.4393,Y -130.4413,Z 165,A -106.7075,B 11.3944,C 0.2908,E1 11.3489,E2 197.4029} C_DIS
LIN {X -39.9914,Y -131.5395,Z 165,A -104.5922,B 11.3947,C 0.2771,E1 11.3548,E2 195.2096} C_DIS
LIN {X -35.7514,Y -132.7549,Z 165,A -103.2061,B 11.3944,C 0.2894,E1 11.3584,E2 193.8812} C_DIS
LIN {X -32.0695,Y -133.6918,Z 165,A -101.6582,B 11.3944,C 0.2912,E1 11.3626,E2 192.3375} C_DIS
LIN {X -28.9276,Y -134.4066,Z 165,A -100.0773,B 11.3944,C 0.286,E1 11.367,E2 190.7258} C_DIS
LIN {X -20.1343,Y -136.0038,Z 165,A -96.4745,B 11.3944,C 0.2904,E1 11.3768,E2 187.1377} C_DIS
LIN {X -15.34,Y -136.627,Z 165,A -94.3682,B 11.3944,C 0.2886,E1 11.3827,E2 185.0189} C_DIS
LIN {X -11.546,Y -136.9988,Z 165,A -92.7164,B 11.3944,C 0.2872,E1 11.3873,E2 183.3584} C_DIS
LIN {X -6.3138,Y -137.3407,Z 165,A -90.7809,B 11.3943,C 0.2935,E1 11.3926,E2 181.454} C_DIS
LIN {X 0.4341,Y -137.4843,Z 165,A -87.975,B 11.3943,C 0.2935,E1 11.4005,E2 178.6478} C_DIS
LIN {X 0.4341,Y -137.4843,Z 165,A -87.975,B 11.3943,C 0.2935,E1 11.4005,E2 178.6478} C_DIS
Enddeposition()
LIN {X 0.9854,Y -138.3876,Z 165,A -87.9599,B 11.0972,C 0.319,E1 11.1038,E2 178.7825} C_DIS
Startdeposition()
$VEL.CP = VEL_PRINT
LIN {X -4.1446,Y -138.3409,Z 165,A -90.3659,B 11.097,C 0.3262,E1 11.097,E2 181.2261} C_DIS
LIN {X -7.6295,Y -138.1939,Z 165,A -91.8609,B 11.097,C 0.3274,E1 11.0928,E2 182.7283} C_DIS
LIN {X -11.3464,Y -137.937,Z 165,A -93.5455,B 11.0968,C 0.3308,E1 11.088,E2 184.4316} C_DIS
LIN {X -18.4708,Y -137.1653,Z 165,A -96.316,B 11.097,C 0.3254,E1 11.0804,E2 187.1782} C_DIS
LIN {X -22.0433,Y -136.6378,Z 165,A -98.2022,B 11.0967,C 0.3343,E1 11.0751,E2 189.1146} C_DIS
LIN {X -25.6138,Y -136.0122,Z 165,A -99.8221,B 11.0967,C 0.3365,E1 11.0706,E2 190.7499} C_DIS
LIN {X -30.006,Y -135.113,Z 165,A -101.178,B 11.097,C 0.3237,E1 11.067,E2 192.043} C_DIS
LIN {X -32.8717,Y -134.4428,Z 165,A -102.4032,B 11.097,C 0.3232,E1 11.0637,E2 193.2692} C_DIS
LIN {X -38.447,Y -132.9548,Z 165,A -104.9331,B 11.097,C 0.325,E1 11.0569,E2 195.8175} C_DIS
LIN {X -42.3945,Y -131.7497,Z 165,A -106.5492,B 11.0971,C 0.3215,E1 11.0526,E2 197.4221} C_DIS
LIN {X -45.6108,Y -130.671,Z 165,A -107.912,B 11.0971,C 0.3194,E1 11.049,E2 198.7798} C_DIS
LIN {X -49.0404,Y -129.4237,Z 165,A -109.4621,B 11.0971,C 0.3189,E1 11.0449,E2 200.3351} C_DIS
LIN {X -52.5316,Y -128.0481,Z 165,A -111.0132,B 11.0972,C 0.3174,E1 11.0409,E2 201.886} C_DIS
LIN {X -55.8087,Y -126.6536,Z 165,A -112.9269,B 11.097,C 0.326,E1 11.0359,E2 203.8553} C_DIS
LIN {X -59.3817,Y -125.0162,Z 165,A -113.9275,B 11.0974,C 0.3097,E1 11.0335,E2 204.7766} C_DIS
LIN {X -63.4556,Y -123.0004,Z 165,A -116.1723,B 11.0973,C 0.3158,E1 11.0278,E2 207.0674} C_DIS
LIN {X -67.636,Y -120.7523,Z 165,A -118.0866,B 11.0973,C 0.3121,E1 11.0231,E2 208.9751} C_DIS
LIN {X -71.4388,Y -118.5422,Z 165,A -119.9267,B 11.0974,C 0.31,E1 11.0187,E2 210.8174} C_DIS
LIN {X -75.2349,Y -116.1699,Z 165,A -121.7823,B 11.0975,C 0.3073,E1 11.0143,E2 212.6731} C_DIS
LIN {X -78.8369,Y -113.7563,Z 165,A -123.6175,B 11.0975,C 0.3054,E1 11.0101,E2 214.5131} C_DIS
LIN {X -82.9329,Y -110.8059,Z 165,A -125.6933,B 11.0977,C 0.3017,E1 11.0054,E2 216.5866} C_DIS
LIN {X -86.5125,Y -108.0345,Z 165,A -127.6199,B 11.0977,C 0.2996,E1 11.0012,E2 218.5193} C_DIS
LIN {X -92.2761,Y -103.1544,Z 165,A -130.6165,B 11.0979,C 0.2911,E1 10.9949,E2 221.4985} C_DIS
LIN {X -95.131,Y -100.5278,Z 165,A -132.3789,B 11.0979,C 0.2915,E1 10.9912,E2 223.2801} C_DIS
LIN {X -98.4298,Y -97.3005,Z 165,A -134.2644,B 11.098,C 0.2871,E1 10.9875,E2 225.1617} C_DIS
LIN {X -101.4996,Y -94.0937,Z 165,A -136.4949,B 11.098,C 0.2919,E1 10.9831,E2 227.4407} C_DIS
LIN {X -104.1992,Y -91.0943,Z 165,A -137.9401,B 11.0981,C 0.2835,E1 10.9805,E2 228.8569} C_DIS
LIN {X -106.795,Y -88.0375,Z 165,A -139.5178,B 11.0983,C 0.278,E1 10.9777,E2 230.4235} C_DIS
LIN {X -109.6635,Y -84.4382,Z 165,A -141.5544,B 11.0983,C 0.2766,E1 10.9742,E2 232.4755} C_DIS
LIN {X -113.0183,Y -79.891,Z 165,A -143.7797,B 11.0985,C 0.2688,E1 10.9706,E2 234.6852} C_DIS
LIN {X -116.6527,Y -74.4841,Z 165,A -146.3477,B 11.0987,C 0.2595,E1 10.9666,E2 237.2354} C_DIS
LIN {X -118.4987,Y -71.5106,Z 165,A -147.9853,B 11.0987,C 0.2601,E1 10.9642,E2 238.8957} C_DIS
LIN {X -120.7577,Y -67.6263,Z 165,A -149.8623,B 11.0987,C 0.2558,E1 10.9616,E2 240.7737} C_DIS
LIN {X -122.7756,Y -63.887,Z 165,A -151.5532,B 11.0989,C 0.2498,E1 10.9594,E2 242.4547} C_DIS
LIN {X -124.167,Y -61.1367,Z 165,A -152.907,B 11.0989,C 0.2482,E1 10.9577,E2 243.8174} C_DIS
LIN {X -125.787,Y -57.7316,Z 165,A -154.4334,B 11.0991,C 0.2434,E1 10.9559,E2 245.3383} C_DIS
LIN {X -127.1567,Y -54.6481,Z 165,A -155.8824,B 11.0991,C 0.2408,E1 10.9543,E2 246.7927} C_DIS
LIN {X -128.8408,Y -50.5511,Z 165,A -158.026,B 11.0991,C 0.2424,E1 10.952,E2 248.9735} C_DIS
LIN {X -130.051,Y -47.3507,Z 165,A -159.0611,B 11.0993,C 0.2305,E1 10.9511,E2 249.9599} C_DIS
LIN {X -131.1707,Y -44.1546,Z 165,A -160.6081,B 11.0993,C 0.2297,E1 10.9496,E2 251.5239} C_DIS
LIN {X -132.3856,Y -40.3642,Z 165,A -163.1019,B 11.0991,C 0.2428,E1 10.9476,E2 254.1211} C_DIS
LIN {X -134.105,Y -34.2212,Z 165,A -164.6547,B 11.0997,C 0.2127,E1 10.9465,E2 255.5367} C_DIS
LIN {X -134.7489,Y -31.6004,Z 165,A -166.2183,B 11.0996,C 0.2189,E1 10.9455,E2 257.1551} C_DIS
LIN {X -135.6547,Y -27.4421,Z 165,A -167.8083,B 11.0997,C 0.2103,E1 10.9446,E2 258.722} C_DIS
LIN {X -136.2751,Y -24.1741,Z 165,A -169.2274,B 11.0997,C 0.2072,E1 10.9438,E2 260.1451} C_DIS
LIN {X -136.9459,Y -20.0319,Z 165,A -171.0262,B 11.0999,C 0.2035,E1 10.9431,E2 261.95} C_DIS
LIN {X -137.4286,Y -16.39,Z 165,A -172.5644,B 11.0999,C 0.1994,E1 10.9425,E2 263.4887} C_DIS
LIN {X -137.8183,Y -12.7139,Z 165,A -174.1922,B 11.0999,C 0.197,E1 10.9421,E2 265.1272} C_DIS
LIN {X -138.1379,Y -8.5569,Z 165,A -175.8671,B 11.1001,C 0.1909,E1 10.9418,E2 266.7941} C_DIS
LIN {X -138.3229,Y -4.7437,Z 165,A -177.5534,B 11.1001,C 0.1885,E1 10.9416,E2 268.4919} C_DIS
LIN {X -138.3833,Y 2.3182,Z 165,A 179.6065,B 11.1003,C 0.1782,E1 10.9416,E2 271.3186} C_DIS
LIN {X -138.2671,Y 6.1723,Z 165,A 177.6843,B 11.1003,C 0.1802,E1 10.9418,E2 273.2796} C_DIS
LIN {X -138.0802,Y 9.4622,Z 165,A 176.5478,B 11.1003,C 0.1715,E1 10.942,E2 274.3864} C_DIS
LIN {X -137.7594,Y 13.3281,Z 165,A 174.9951,B 11.1005,C 0.1657,E1 10.9424,E2 275.9307} C_DIS
LIN {X -137.3674,Y 16.9035,Z 165,A 173.4155,B 11.1005,C 0.1632,E1 10.9429,E2 277.52} C_DIS
LIN {X -136.8107,Y 20.9319,Z 165,A 171.7543,B 11.1005,C 0.1578,E1 10.9435,E2 279.1766} C_DIS
LIN {X -136.218,Y 24.4932,Z 165,A 170.2076,B 11.1006,C 0.1546,E1 10.9443,E2 280.7281} C_DIS
LIN {X -135.5914,Y 27.7528,Z 165,A 168.8983,B 11.1007,C 0.1492,E1 10.945,E2 282.0279} C_DIS
LIN {X -134.8695,Y 31.0726,Z 165,A 167.4227,B 11.1007,C 0.1466,E1 10.9459,E2 283.5105} C_DIS
LIN {X -134.0232,Y 34.5433,Z 165,A 165.8647,B 11.1007,C 0.144,E1 10.9469,E2 285.0765} C_DIS
LIN {X -132.9936,Y 38.3177,Z 165,A 164.1882,B 11.1008,C 0.1406,E1 10.9482,E2 286.7583} C_DIS
LIN {X -131.7069,Y 42.5285,Z 165,A 161.9373,B 11.1008,C 0.1443,E1 10.9502,E2 289.0598} C_DIS
LIN {X -130.2881,Y 46.6933,Z 165,A 159.7526,B 11.1008,C 0.1467,E1 10.9523,E2 291.2867} C_DIS
LIN {X -128.0185,Y 52.6029,Z 165,A 157.9677,B 11.101,C 0.1222,E1 10.954,E2 292.9664} C_DIS
Enddeposition()
END
